	WAMANAGER_CICLO_DEPOSITO_FALDA_VUOTI_RUN:
		DirezioneXPositiva := TFDirezioneAssePositiva(Posizione_Attuale:=ModuleAX_X^.Ax^.Status.ActPosition,Posizione_Finale:=Mission^.XPlace);
		DirezioneXNegativa := NOT DirezioneXPositiva;
		(* Valuto se con l'asse X sono fuori dall'area delle colonne *)
		QuotaX_ConsensoRotazionePinza_Raggiunta := TFPinzaInFuoriIngombroColonne_DirezioneX(DirezioneXPositiva:=DirezioneXPositiva,
																							AsseInMoto:=ModuleAX_X^.Ax^.AxRef^.Status.Moving,
																							PosizioneAttuale:=ModuleAX_X^.Ax^.Status.ActPosition,
																							PosizioneColonna_X:=WorkFootprint^[5].X,  
																							IngombroColonna_X:=WorkFootprint^[5].XDim,
																							IngombroPinza_X:=IngombroX);
				IF CalcolaIngombro THEN
			CalcolaIngombro := FALSE;
			(* Definisco il tipo di area in cui si trova a lavorare il pallettizzatore *)
			AreaInLavoroPositiva := FALSE;
			AreaInLavoroNegativa := FALSE;
			AreaInLavoroPositivaNegativa := FALSE; 
			
			IF (WorkArea^[Mission^.PPlace].X >= (WorkFootprint^[5].X + WorkFootprint^[5].XDim)) AND 		//se la piazzola di prelievo è nella campata POSITIVA
				(ModuleAX_X^.Ax^.Status.ActPosition >= (WorkFootprint^[5].X + WorkFootprint^[5].XDim)) THEN // Se la posizione attuale è nella campata POSITIVA
					AreaInLavoroPositivaNegativa := FALSE; 
					AreaInLavoroPositiva := TRUE;
			ELSIF (WorkArea^[Mission^.PPlace].X <= WorkFootprint^[5].X) AND 			//se la piazzola di prelievo è nella campata NEGATIVA
				(ModuleAX_X^.Ax^.Status.ActPosition <= WorkFootprint^[5].X) THEN 		// Se la posizione attuale è nella campata NEGATIVA
					AreaInLavoroPositivaNegativa := FALSE; 
					AreaInLavoroNegativa := TRUE;
			ELSE
				AreaInLavoroPositivaNegativa := TRUE;
			END_IF
			
			(**************************************************************************************************************************************************)
			(* Ingombro ottimizzato della pinza sul punto di prelievo *)
			(**************************************************************************************************************************************************)
			IngombroOttimizzatoX_InPuntoDiPrelievo := ABS(IngombroSuperficialePinzaMAX * SIN(deg_to_rad((ATAN(Larghezza/Lunghezza)*1/0.017+ Mission^.JPick))));
			IngombroOttimizzatoY_InPuntoDiPrelievo := ABS(IngombroSuperficialePinzaMAX * COS(deg_to_rad((ATAN(Larghezza/Lunghezza)*1/0.017+ Mission^.JPick))));
			(**************************************************************************************************************************************************)
			(* Ingombro ottimizzato della pinza sul punto di deposito *)
			(**************************************************************************************************************************************************)
			IngombroOttimizzatoX_InPuntoDiDeposito := ABS(IngombroSuperficialePinzaMAX * SIN(deg_to_rad((ATAN(Larghezza/Lunghezza)*1/0.017+ Mission^.JPlace))));
			IngombroOttimizzatoY_InPuntoDiDeposito := ABS(IngombroSuperficialePinzaMAX * COS(deg_to_rad((ATAN(Larghezza/Lunghezza)*1/0.017+ Mission^.JPlace))));
						
			(**************************************************************************************************************************************************)
			(**************************************************************************************************************************************************)
			(* Valuto la direzione della X *)
			DirezioneXPositiva := TFDirezioneAssePositiva(Posizione_Attuale:=ModuleAX_X^.Ax^.Status.ActPosition,Posizione_Finale:=Mission^.XPlace);
			DirezioneXNegativa := NOT DirezioneXPositiva;
							
			(**************************************************************************************************************************************************)
			(* Ingombro MASSIMO della pinza durante il transito *)
			(**************************************************************************************************************************************************)
			//Calcolo ingombro attuale
			IF NOT TFAsseInFinestra(Posizione_Attuale:=ModuleAx_J^.Ax^.AxRef^.NcToPlc.ActPos,Posizione_Finale:=Mission^.JPlace,FinestraDiControllo:=5)  THEN //Se la pinza non è già nella finestra di destinazione 
				(* Calcolo l'ingombro massimo che assume durante il ciclo di lavoro nelle direzioni X e Y *)
				TFCalcoloIngombroOttimizzatoPinza(  Quota_RotazioneAttuale			:= ModuleAx_J^.Ax^.AxRef^.NcToPlc.ActPos,
													Quota_RotazioneDestinazione		:= Mission^.JPlace,
													IngombroSuperficialePinzaMAX	:= IngombroSuperficialePinzaMAX,
													Lunghezza						:= Larghezza,
													Larghezza						:= Lunghezza,
													IngombroOttimizzatoX_InTransito	=> IngombroOttimizzatoX_InTransito,
													IngombroOttimizzatoY_InTransito	=> IngombroOttimizzatoY_InTransito);
			ELSE
				IngombroOttimizzatoX_InTransito := ABS(IngombroSuperficialePinzaMAX * SIN(deg_to_rad((ATAN(Larghezza/Lunghezza)*1/0.017+ ModuleAx_J^.Ax^.AxRef^.NcToPlc.ActPos)))); //Ingombro Attuale direzione X
				IngombroOttimizzatoY_InTransito := ABS(IngombroSuperficialePinzaMAX * COS(deg_to_rad((ATAN(Larghezza/Lunghezza)*1/0.017+ ModuleAx_J^.Ax^.AxRef^.NcToPlc.ActPos)))); //Ingombro Attuale direzione Y		
			END_IF
			(* Valutazione colonne in base al verso del pallettizzatore: verso stabilito guardando il pallettizzatore con la linea alle spalle *)
			CASE VERSO_PALLETTIZZATORE OF
				PALLETTIZZATORE_DX :
									TFCalcolaQuotaIngombroColonne(	QuotaY_ColonnaDX						:= WorkFootprint^[6].Y, //DX
																	QuotaY_ColonnaSX						:= WorkFootprint^[5].Y, //SX
																	QuotaAttualeAsse						:= ModuleAX_Y^.Ax^.AxRef^.NcToPlc.ActPos,
																	IngombroOttimizzatoY_InTransito         := IngombroOttimizzatoY_InTransito,
																	OffsetSicurezza_Y						:= OffsetSicurezza_Y,
																	QuotaDestinazioneAsse					:= Mission^.YPlace,
																	Pinza_InIngombroColonne_Attuale 		=> Pinza_InIngombroColonne_Attuale,
																	Pinza_InIngombroColonne_Destinazione 	=> Pinza_InIngombroColonne_Destinazione,
																	QuotaFuoriIngombro_Attuale_Y 			=> QuotaFuoriIngombro_Attuale_Y,
																	QuotaFuoriIngombro_Destinazione_Y 		=> QuotaFuoriIngombro_Destinazione_Y);
																	
				PALLETTIZZATORE_SX :
									TFCalcolaQuotaIngombroColonne(	QuotaY_ColonnaDX						:= WorkFootprint^[6].Y, //DX
																	QuotaY_ColonnaSX						:= WorkFootprint^[5].Y, //SX
																	QuotaAttualeAsse						:= ModuleAX_Y^.Ax^.AxRef^.NcToPlc.ActPos,
																	OffsetSicurezza_Y						:= OffsetSicurezza_Y,
																	IngombroOttimizzatoY_InTransito         := IngombroOttimizzatoY_InTransito,
																	QuotaDestinazioneAsse					:= Mission^.YPlace,
																	Pinza_InIngombroColonne_Attuale 		=> Pinza_InIngombroColonne_Attuale,
																	Pinza_InIngombroColonne_Destinazione 	=> Pinza_InIngombroColonne_Destinazione,
																	QuotaFuoriIngombro_Attuale_Y 			=> QuotaFuoriIngombro_Attuale_Y,
																	QuotaFuoriIngombro_Destinazione_Y 		=> QuotaFuoriIngombro_Destinazione_Y);
			END_CASE
			
			(* Setto la quota di fuori ingombro che la pinza dovrà assumere durante la traslazione per evitare la collisione con le colonne *)	
			QuotaFuoriIngombroColonne_Y := MAX(QuotaFuoriIngombro_Attuale_Y,QuotaFuoriIngombro_Destinazione_Y);
					
			(* Se sono in ingombro nella posizione attuale o nella posizione di destinazione, devo andare fuori-ingombro con la Y *)
			IF (Pinza_InIngombroColonne_Attuale OR Pinza_InIngombroColonne_Destinazione) THEN 
				IF (AsseXInFinestraDiRiposo AND AsseYInFinestraDiRiposo AND AsseJInFinestraDiRiposo) THEN //Se sono in finestra di riposo con tutti gli assi non devo andare fuori-ingombro con la Y
					FuoriIngombroYNecessarioTMP := FALSE;
				ELSE
					FuoriIngombroYNecessarioTMP := TRUE;
				END_IF
			ELSE
				FuoriIngombroYNecessarioTMP := FALSE;
			END_IF
		END_IF
								
	//WAMANAGER_CICLO_DEPOSITO_FALDA_VUOTI_END:
	//	CalcolaIngombro := TRUE;	
	*)
	WAMANAGER_CICLO_FALDA_INIT:
		CalcolaIngombro := TRUE;	
	
	WAMANAGER_CICLO_PRELIEVO_FALDA_RUN:
		DirezioneXPositiva := TFDirezioneAssePositiva(Posizione_Attuale:=ModuleAX_X^.Ax^.Status.ActPosition,Posizione_Finale:=Mission^.XPick);
		DirezioneXNegativa := NOT DirezioneXPositiva;
		(* Valuto se con l'asse X sono fuori dall'area delle colonne *)
		(*QuotaX_ConsensoRotazionePinza_Raggiunta := TFPinzaInFuoriIngombroColonne_DirezioneX(DirezioneXPositiva:=DirezioneXPositiva,
																							AsseInMoto:=ModuleAX_X^.Ax^.AxRef^.Status.Moving,
																							PosizioneAttuale:=ModuleAX_X^.Ax^.Status.ActPosition,
																							PosizioneColonna_X:=WorkFootprint^[5].X,  
																							IngombroColonna_X:=WorkFootprint^[5].XDim,
																							IngombroPinza_X:=IngombroX);*)
																							
		IF CalcolaIngombro THEN
			CalcolaIngombro := FALSE;
			(* Definisco il tipo di area in cui si trova a lavorare il pallettizzatore *)
			AreaInLavoroPositiva := FALSE;
			AreaInLavoroNegativa := FALSE;
			AreaInLavoroPositivaNegativa := FALSE; 
			
			IF (WorkArea^[Mission^.PPick].X >= (WorkFootprint^[5].X + WorkFootprint^[5].XDim)) AND 				//se la piazzola di prelievo è nella campata POSITIVA
				(ModuleAX_X^.Ax^.Status.ActPosition >= (WorkFootprint^[5].X + WorkFootprint^[5].XDim)) THEN // Se la posizione attuale è nella campata POSITIVA
					AreaInLavoroPositiva := TRUE;
			ELSIF (WorkArea^[Mission^.PPick].X <= WorkFootprint^[5].X) AND 			//se la piazzola di prelievo è nella campata NEGATIVA
				(ModuleAX_X^.Ax^.Status.ActPosition <= WorkFootprint^[5].X) THEN 		// Se la posizione attuale è nella campata NEGATIVA
					AreaInLavoroNegativa := TRUE;
			ELSE
				AreaInLavoroPositivaNegativa := TRUE;
			END_IF
			(**************************************************************************************************************************************************)
			(* Ingombro ottimizzato della pinza sul punto di prelievo *)
			(**************************************************************************************************************************************************)
			(*IngombroOttimizzatoX_InPuntoDiPrelievo := ABS(IngombroSuperficialePinzaMAX * SIN(deg_to_rad((ATAN(Larghezza/Lunghezza)*1/0.017+ Mission^.JPick))));
			IngombroOttimizzatoY_InPuntoDiPrelievo := ABS(IngombroSuperficialePinzaMAX * COS(deg_to_rad((ATAN(Larghezza/Lunghezza)*1/0.017+ Mission^.JPick))));
			(**************************************************************************************************************************************************)
			(* Ingombro ottimizzato della pinza sul punto di deposito *)
			(**************************************************************************************************************************************************)
			IngombroOttimizzatoX_InPuntoDiDeposito := ABS(IngombroSuperficialePinzaMAX * SIN(deg_to_rad((ATAN(Larghezza/Lunghezza)*1/0.017+ Mission^.JPlace))));
			IngombroOttimizzatoY_InPuntoDiDeposito := ABS(IngombroSuperficialePinzaMAX * COS(deg_to_rad((ATAN(Larghezza/Lunghezza)*1/0.017+ Mission^.JPlace))));
			*)			
			(**************************************************************************************************************************************************)
			(**************************************************************************************************************************************************)
			(* Valuto la direzione della X *)
			DirezioneXPositiva := TFDirezioneAssePositiva(Posizione_Attuale:=ModuleAX_X^.Ax^.Status.ActPosition,Posizione_Finale:=Mission^.XPick);
			DirezioneXNegativa := NOT DirezioneXPositiva;
							
			(**************************************************************************************************************************************************)
			(* Ingombro MASSIMO della pinza durante il transito *)
			(**************************************************************************************************************************************************)
			//Calcolo ingombro attuale
			IF NOT TFAsseInFinestra(Posizione_Attuale:=ModuleAx_J^.Ax^.AxRef^.NcToPlc.ActPos,Posizione_Finale:=Mission^.JPick,FinestraDiControllo:=5)  THEN //Se la pinza non è già nella finestra di destinazione 
				(* Calcolo l'ingombro massimo che assume durante il ciclo di lavoro nelle direzioni X e Y *)
				(*TFCalcoloIngombroOttimizzatoPinza(  Quota_RotazioneAttuale			:= ModuleAx_J^.Ax^.AxRef^.NcToPlc.ActPos,
													Quota_RotazioneDestinazione		:= Mission^.JPick,
													IngombroSuperficialePinzaMAX	:= IngombroSuperficialePinzaMAX,
													Lunghezza						:= Larghezza,
													Larghezza						:= Lunghezza,
													IngombroOttimizzatoX_InTransito	=> IngombroOttimizzatoX_InTransito,
													IngombroOttimizzatoY_InTransito	=> IngombroOttimizzatoY_InTransito);*)
			ELSE;
				//IngombroOttimizzatoX_InTransito := ABS(IngombroSuperficialePinzaMAX * SIN(deg_to_rad((ATAN(Larghezza/Lunghezza)*1/0.017+ ModuleAx_J^.Ax^.AxRef^.NcToPlc.ActPos)))); //Ingombro Attuale direzione X
				//IngombroOttimizzatoY_InTransito := ABS(IngombroSuperficialePinzaMAX * COS(deg_to_rad((ATAN(Larghezza/Lunghezza)*1/0.017+ ModuleAx_J^.Ax^.AxRef^.NcToPlc.ActPos)))); //Ingombro Attuale direzione Y		
			END_IF
			(* Valutazione colonne in base al verso del pallettizzatore: verso stabilito guardando il pallettizzatore con la linea alle spalle *)
			CASE VERSO_PALLETTIZZATORE OF
				PALLETTIZZATORE_DX :
									TFCalcolaQuotaIngombroColonne(	QuotaY_ColonnaDX						:= WorkFootprint^[6].Y, //DX
																	QuotaY_ColonnaSX						:= WorkFootprint^[5].Y, //SX
																	QuotaAttualeAsse						:= ModuleAX_Y^.Ax^.AxRef^.NcToPlc.ActPos,
																	IngombroOttimizzatoY_InTransito         := IngombroOttimizzatoY_InTransito,
																	OffsetSicurezza_Y						:= OffsetSicurezza_Y,
																	QuotaDestinazioneAsse					:= Mission^.YPick,
																	Pinza_InIngombroColonne_Attuale 		=> Pinza_InIngombroColonne_Attuale,
																	Pinza_InIngombroColonne_Destinazione 	=> Pinza_InIngombroColonne_Destinazione,
																	QuotaFuoriIngombro_Attuale_Y 			=> QuotaFuoriIngombro_Attuale_Y,
																	QuotaFuoriIngombro_Destinazione_Y 		=> QuotaFuoriIngombro_Destinazione_Y);
																	
				PALLETTIZZATORE_SX :
									TFCalcolaQuotaIngombroColonne(	QuotaY_ColonnaDX						:= WorkFootprint^[6].Y, //DX
																	QuotaY_ColonnaSX						:= WorkFootprint^[5].Y, //SX
																	QuotaAttualeAsse						:= ModuleAX_Y^.Ax^.AxRef^.NcToPlc.ActPos,
																	OffsetSicurezza_Y						:= OffsetSicurezza_Y,
																	IngombroOttimizzatoY_InTransito         := IngombroOttimizzatoY_InTransito,
																	QuotaDestinazioneAsse					:= Mission^.YPick,
																	Pinza_InIngombroColonne_Attuale 		=> Pinza_InIngombroColonne_Attuale,
																	Pinza_InIngombroColonne_Destinazione 	=> Pinza_InIngombroColonne_Destinazione,
																	QuotaFuoriIngombro_Attuale_Y 			=> QuotaFuoriIngombro_Attuale_Y,
																	QuotaFuoriIngombro_Destinazione_Y 		=> QuotaFuoriIngombro_Destinazione_Y);
			END_CASE
			
			(* Setto la quota di fuori ingombro che la pinza dovrà assumere durante la traslazione per evitare la collisione con le colonne *)	
			QuotaFuoriIngombroColonne_Y := QuotaFuoriIngombro_Attuale_Y;
					
			(* Se sono in ingombro nella posizione attuale o nella posizione di destinazione, devo andare fuori-ingombro con la Y *)
			IF (Pinza_InIngombroColonne_Attuale OR Pinza_InIngombroColonne_Destinazione) THEN 
				IF (AsseXInFinestraDiRiposo AND AsseYInFinestraDiRiposo AND AsseJInFinestraDiRiposo) THEN //Se sono in finestra di riposo con tutti gli assi non devo andare fuori-ingombro con la Y
					FuoriIngombroYNecessarioTMP := FALSE;
				ELSE
					FuoriIngombroYNecessarioTMP := TRUE;
				END_IF
			ELSE
				FuoriIngombroYNecessarioTMP := FALSE;
			END_IF
		END_IF	
																
	WAMANAGER_CICLO_PRELIEVO_FALDA_END:
		CalcolaIngombro := TRUE;	
			
	WAMANAGER_CICLO_DEPOSITO_FALDA_RUN:
		DirezioneXPositiva := TFDirezioneAssePositiva(Posizione_Attuale:=ModuleAX_X^.Ax^.Status.ActPosition,Posizione_Finale:=Mission^.XPlace);
		DirezioneXNegativa := NOT DirezioneXPositiva;
		(* Valuto se con l'asse X sono fuori dall'area delle colonne *)
		(*QuotaX_ConsensoRotazionePinza_Raggiunta := TFPinzaInFuoriIngombroColonne_DirezioneX(DirezioneXPositiva:=DirezioneXPositiva,
																							AsseInMoto:=ModuleAX_X^.Ax^.AxRef^.Status.Moving,
																							PosizioneAttuale:=ModuleAX_X^.Ax^.Status.ActPosition,
																							PosizioneColonna_X:=WorkFootprint^[5].X,  
																							IngombroColonna_X:=WorkFootprint^[5].XDim,
																							IngombroPinza_X:=IngombroX);*)
																							
		IF (WorkArea^[Mission^.PPlace].X >= (WorkFootprint^[5].X + WorkFootprint^[5].XDim)) AND 				//se la piazzola di prelievo è nella campata POSITIVA
			(ModuleAX_X^.Ax^.Status.ActPosition >= (WorkFootprint^[5].X + WorkFootprint^[5].XDim)) THEN // Se la posizione attuale è nella campata POSITIVA
				AreaInLavoroPositiva := TRUE;
		ELSIF (WorkArea^[Mission^.PPlace].X <= WorkFootprint^[5].X) AND 			//se la piazzola di prelievo è nella campata NEGATIVA
			(ModuleAX_X^.Ax^.Status.ActPosition <= WorkFootprint^[5].X) THEN 		// Se la posizione attuale è nella campata NEGATIVA
				AreaInLavoroNegativa := TRUE;
		ELSE
			AreaInLavoroPositivaNegativa := TRUE;
		END_IF
		
		IF CalcolaIngombro THEN
			CalcolaIngombro := FALSE;
			(* Definisco il tipo di area in cui si trova a lavorare il pallettizzatore *)
			AreaInLavoroPositiva := FALSE;
			AreaInLavoroNegativa := FALSE;
			AreaInLavoroPositivaNegativa := TRUE; 
			
			(**************************************************************************************************************************************************)
			(* Ingombro ottimizzato della pinza sul punto di prelievo *)
			(**************************************************************************************************************************************************)
		(*	IngombroOttimizzatoX_InPuntoDiPrelievo := ABS(IngombroSuperficialePinzaMAX * SIN(deg_to_rad((ATAN(Larghezza/Lunghezza)*1/0.017+ Mission^.JPick))));
			IngombroOttimizzatoY_InPuntoDiPrelievo := ABS(IngombroSuperficialePinzaMAX * COS(deg_to_rad((ATAN(Larghezza/Lunghezza)*1/0.017+ Mission^.JPick))));
			(**************************************************************************************************************************************************)
			(* Ingombro ottimizzato della pinza sul punto di deposito *)
			(**************************************************************************************************************************************************)
			IngombroOttimizzatoX_InPuntoDiDeposito := ABS(IngombroSuperficialePinzaMAX * SIN(deg_to_rad((ATAN(Larghezza/Lunghezza)*1/0.017+ Mission^.JPlace))));
			IngombroOttimizzatoY_InPuntoDiDeposito := ABS(IngombroSuperficialePinzaMAX * COS(deg_to_rad((ATAN(Larghezza/Lunghezza)*1/0.017+ Mission^.JPlace))));
			*)			
			(**************************************************************************************************************************************************)
			(**************************************************************************************************************************************************)
			(* Valuto la direzione della X *)
			DirezioneXPositiva := TFDirezioneAssePositiva(Posizione_Attuale:=ModuleAX_X^.Ax^.Status.ActPosition,Posizione_Finale:=Mission^.XPlace);
			DirezioneXNegativa := NOT DirezioneXPositiva;
							
			(**************************************************************************************************************************************************)
			(* Ingombro MASSIMO della pinza durante il transito *)
			(**************************************************************************************************************************************************)
			//Calcolo ingombro attuale
			IF NOT TFAsseInFinestra(Posizione_Attuale:=ModuleAx_J^.Ax^.AxRef^.NcToPlc.ActPos,Posizione_Finale:=Mission^.JPlace,FinestraDiControllo:=5)  THEN //Se la pinza non è già nella finestra di destinazione 
				(* Calcolo l'ingombro massimo che assume durante il ciclo di lavoro nelle direzioni X e Y *)
				(*TFCalcoloIngombroOttimizzatoPinza(  Quota_RotazioneAttuale			:= ModuleAx_J^.Ax^.AxRef^.NcToPlc.ActPos,
													Quota_RotazioneDestinazione		:= Mission^.JPlace,
													IngombroSuperficialePinzaMAX	:= IngombroSuperficialePinzaMAX,
													Lunghezza						:= Larghezza,
													Larghezza						:= Lunghezza,
													IngombroOttimizzatoX_InTransito	=> IngombroOttimizzatoX_InTransito,
													IngombroOttimizzatoY_InTransito	=> IngombroOttimizzatoY_InTransito);*)
			ELSE;
				//IngombroOttimizzatoX_InTransito := ABS(IngombroSuperficialePinzaMAX * SIN(deg_to_rad((ATAN(Larghezza/Lunghezza)*1/0.017+ ModuleAx_J^.Ax^.AxRef^.NcToPlc.ActPos)))); //Ingombro Attuale direzione X
				//IngombroOttimizzatoY_InTransito := ABS(IngombroSuperficialePinzaMAX * COS(deg_to_rad((ATAN(Larghezza/Lunghezza)*1/0.017+ ModuleAx_J^.Ax^.AxRef^.NcToPlc.ActPos)))); //Ingombro Attuale direzione Y		
			END_IF
			(* Valutazione colonne in base al verso del pallettizzatore: verso stabilito guardando il pallettizzatore con la linea alle spalle *)
			CASE VERSO_PALLETTIZZATORE OF
				PALLETTIZZATORE_DX :
									TFCalcolaQuotaIngombroColonne(	QuotaY_ColonnaDX						:= WorkFootprint^[6].Y, //DX
																	QuotaY_ColonnaSX						:= WorkFootprint^[5].Y, //SX
																	QuotaAttualeAsse						:= ModuleAX_Y^.Ax^.AxRef^.NcToPlc.ActPos,
																	IngombroOttimizzatoY_InTransito         := IngombroOttimizzatoY_InTransito,
																	OffsetSicurezza_Y						:= OffsetSicurezza_Y,
																	QuotaDestinazioneAsse					:= Mission^.YPlace,
																	Pinza_InIngombroColonne_Attuale 		=> Pinza_InIngombroColonne_Attuale,
																	Pinza_InIngombroColonne_Destinazione 	=> Pinza_InIngombroColonne_Destinazione,
																	QuotaFuoriIngombro_Attuale_Y 			=> QuotaFuoriIngombro_Attuale_Y,
																	QuotaFuoriIngombro_Destinazione_Y 		=> QuotaFuoriIngombro_Destinazione_Y);
																	
				PALLETTIZZATORE_SX :
									TFCalcolaQuotaIngombroColonne(	QuotaY_ColonnaDX						:= WorkFootprint^[6].Y, //DX
																	QuotaY_ColonnaSX						:= WorkFootprint^[5].Y, //SX
																	QuotaAttualeAsse						:= ModuleAX_Y^.Ax^.AxRef^.NcToPlc.ActPos,
																	OffsetSicurezza_Y						:= OffsetSicurezza_Y,
																	IngombroOttimizzatoY_InTransito         := IngombroOttimizzatoY_InTransito,
																	QuotaDestinazioneAsse					:= Mission^.YPlace,
																	Pinza_InIngombroColonne_Attuale 		=> Pinza_InIngombroColonne_Attuale,
																	Pinza_InIngombroColonne_Destinazione 	=> Pinza_InIngombroColonne_Destinazione,
																	QuotaFuoriIngombro_Attuale_Y 			=> QuotaFuoriIngombro_Attuale_Y,
																	QuotaFuoriIngombro_Destinazione_Y 		=> QuotaFuoriIngombro_Destinazione_Y);
			END_CASE
			
			(* Setto la quota di fuori ingombro che la pinza dovrà assumere durante la traslazione per evitare la collisione con le colonne *)	
			QuotaFuoriIngombroColonne_Y := QuotaFuoriIngombro_Attuale_Y;
					
			(* Se sono in ingombro nella posizione attuale o nella posizione di destinazione, devo andare fuori-ingombro con la Y *)
			IF (Pinza_InIngombroColonne_Attuale OR Pinza_InIngombroColonne_Destinazione) THEN 
				IF (AsseXInFinestraDiRiposo AND AsseYInFinestraDiRiposo AND AsseJInFinestraDiRiposo) THEN //Se sono in finestra di riposo con tutti gli assi non devo andare fuori-ingombro con la Y
					FuoriIngombroYNecessarioTMP := FALSE;
				ELSE
					FuoriIngombroYNecessarioTMP := TRUE;
				END_IF
			ELSE
				FuoriIngombroYNecessarioTMP := FALSE;
			END_IF
		END_IF
			
	WAMANAGER_CICLO_DEPOSITO_FALDA_END:
		CalcolaIngombro := TRUE;	
(*
	WAMANAGER_CICLO_PACCO_INIT:
		CalcolaIngombro := TRUE;	
	
	WAMANAGER_CICLO_PRELIEVO_PACCO_RUN:
		DirezioneXPositiva := TFDirezioneAssePositiva(Posizione_Attuale:=ModuleAX_X^.Ax^.Status.ActPosition,Posizione_Finale:=Mission^.XPick);
		DirezioneXNegativa := NOT DirezioneXPositiva;
		(* Valuto se con l'asse X sono fuori dall'area delle colonne *)
		QuotaX_ConsensoRotazionePinza_Raggiunta := TFPinzaInFuoriIngombroColonne_DirezioneX(DirezioneXPositiva:=DirezioneXPositiva,
																							AsseInMoto:=ModuleAX_X^.Ax^.AxRef^.Status.Moving,
																							PosizioneAttuale:=ModuleAX_X^.Ax^.Status.ActPosition,
																							PosizioneColonna_X:=WorkFootprint^[5].X,  
																							IngombroColonna_X:=WorkFootprint^[5].XDim,
																							IngombroPinza_X:=IngombroX);																				
		
		IF CalcolaIngombro THEN
			CalcolaIngombro := FALSE;
			(* Definisco il tipo di area in cui si trova a lavorare il pallettizzatore *)
			AreaInLavoroPositiva := FALSE;
			AreaInLavoroNegativa := FALSE;
			AreaInLavoroPositivaNegativa := TRUE; 
			
			(**************************************************************************************************************************************************)
			(* Ingombro ottimizzato della pinza sul punto di prelievo *)
			(**************************************************************************************************************************************************)
			IngombroOttimizzatoX_InPuntoDiPrelievo := ABS(IngombroSuperficialePinzaMAX * SIN(deg_to_rad((ATAN(Larghezza/Lunghezza)*1/0.017+ Mission^.JPick))));
			IngombroOttimizzatoY_InPuntoDiPrelievo := ABS(IngombroSuperficialePinzaMAX * COS(deg_to_rad((ATAN(Larghezza/Lunghezza)*1/0.017+ Mission^.JPick))));
			(**************************************************************************************************************************************************)
			(* Ingombro ottimizzato della pinza sul punto di deposito *)
			(**************************************************************************************************************************************************)
			IngombroOttimizzatoX_InPuntoDiDeposito := ABS(IngombroSuperficialePinzaMAX * SIN(deg_to_rad((ATAN(Larghezza/Lunghezza)*1/0.017+ Mission^.JPlace))));
			IngombroOttimizzatoY_InPuntoDiDeposito := ABS(IngombroSuperficialePinzaMAX * COS(deg_to_rad((ATAN(Larghezza/Lunghezza)*1/0.017+ Mission^.JPlace))));
						
			(**************************************************************************************************************************************************)
			(**************************************************************************************************************************************************)
			(* Valuto la direzione della X *)
			DirezioneXPositiva := TFDirezioneAssePositiva(Posizione_Attuale:=ModuleAX_X^.Ax^.Status.ActPosition,Posizione_Finale:=Mission^.XPick);
			DirezioneXNegativa := NOT DirezioneXPositiva;
							
			(**************************************************************************************************************************************************)
			(* Ingombro MASSIMO della pinza durante il transito *)
			(**************************************************************************************************************************************************)
			//Calcolo ingombro attuale
			IF NOT TFAsseInFinestra(Posizione_Attuale:=ModuleAx_J^.Ax^.AxRef^.NcToPlc.ActPos,Posizione_Finale:=Mission^.JPick,FinestraDiControllo:=5)  THEN //Se la pinza non è già nella finestra di destinazione 
				(* Calcolo l'ingombro massimo che assume durante il ciclo di lavoro nelle direzioni X e Y *)
				TFCalcoloIngombroOttimizzatoPinza(  Quota_RotazioneAttuale			:= ModuleAx_J^.Ax^.AxRef^.NcToPlc.ActPos,
													Quota_RotazioneDestinazione		:= Mission^.JPick,
													IngombroSuperficialePinzaMAX	:= IngombroSuperficialePinzaMAX,
													Lunghezza						:= Larghezza,
													Larghezza						:= Lunghezza,
													IngombroOttimizzatoX_InTransito	=> IngombroOttimizzatoX_InTransito,
													IngombroOttimizzatoY_InTransito	=> IngombroOttimizzatoY_InTransito);
			ELSE
				IngombroOttimizzatoX_InTransito := ABS(IngombroSuperficialePinzaMAX * SIN(deg_to_rad((ATAN(Larghezza/Lunghezza)*1/0.017+ ModuleAx_J^.Ax^.AxRef^.NcToPlc.ActPos)))); //Ingombro Attuale direzione X
				IngombroOttimizzatoY_InTransito := ABS(IngombroSuperficialePinzaMAX * COS(deg_to_rad((ATAN(Larghezza/Lunghezza)*1/0.017+ ModuleAx_J^.Ax^.AxRef^.NcToPlc.ActPos)))); //Ingombro Attuale direzione Y		
			END_IF
			(* Valutazione colonne in base al verso del pallettizzatore: verso stabilito guardando il pallettizzatore con la linea alle spalle *)
			CASE VERSO_PALLETTIZZATORE OF
				PALLETTIZZATORE_DX :
									TFCalcolaQuotaIngombroColonne(	QuotaY_ColonnaDX						:= WorkFootprint^[6].Y, //DX
																	QuotaY_ColonnaSX						:= WorkFootprint^[5].Y, //SX
																	QuotaAttualeAsse						:= ModuleAX_Y^.Ax^.AxRef^.NcToPlc.ActPos,
																	IngombroOttimizzatoY_InTransito         := IngombroOttimizzatoY_InTransito,
																	OffsetSicurezza_Y						:= OffsetSicurezza_Y,
																	QuotaDestinazioneAsse					:= Mission^.YPick,
																	Pinza_InIngombroColonne_Attuale 		=> Pinza_InIngombroColonne_Attuale,
																	Pinza_InIngombroColonne_Destinazione 	=> Pinza_InIngombroColonne_Destinazione,
																	QuotaFuoriIngombro_Attuale_Y 			=> QuotaFuoriIngombro_Attuale_Y,
																	QuotaFuoriIngombro_Destinazione_Y 		=> QuotaFuoriIngombro_Destinazione_Y);
																	
				PALLETTIZZATORE_SX :
									TFCalcolaQuotaIngombroColonne(	QuotaY_ColonnaDX						:= WorkFootprint^[6].Y, //DX
																	QuotaY_ColonnaSX						:= WorkFootprint^[5].Y, //SX
																	QuotaAttualeAsse						:= ModuleAX_Y^.Ax^.AxRef^.NcToPlc.ActPos,
																	OffsetSicurezza_Y						:= OffsetSicurezza_Y,
																	IngombroOttimizzatoY_InTransito         := IngombroOttimizzatoY_InTransito,
																	QuotaDestinazioneAsse					:= Mission^.YPick,
																	Pinza_InIngombroColonne_Attuale 		=> Pinza_InIngombroColonne_Attuale,
																	Pinza_InIngombroColonne_Destinazione 	=> Pinza_InIngombroColonne_Destinazione,
																	QuotaFuoriIngombro_Attuale_Y 			=> QuotaFuoriIngombro_Attuale_Y,
																	QuotaFuoriIngombro_Destinazione_Y 		=> QuotaFuoriIngombro_Destinazione_Y);
			END_CASE
			
			(* Setto la quota di fuori ingombro che la pinza dovrà assumere durante la traslazione per evitare la collisione con le colonne *)	
			QuotaFuoriIngombroColonne_Y := QuotaFuoriIngombro_Attuale_Y;
					
			(* Se sono in ingombro nella posizione attuale o nella posizione di destinazione, devo andare fuori-ingombro con la Y *)
			IF (Pinza_InIngombroColonne_Attuale OR Pinza_InIngombroColonne_Destinazione) THEN 
				IF (AsseXInFinestraDiRiposo AND AsseYInFinestraDiRiposo AND AsseJInFinestraDiRiposo) THEN //Se sono in finestra di riposo con tutti gli assi non devo andare fuori-ingombro con la Y
					FuoriIngombroYNecessarioTMP := FALSE;
				ELSE
					FuoriIngombroYNecessarioTMP := TRUE;
				END_IF
			ELSE
				FuoriIngombroYNecessarioTMP := FALSE;
			END_IF
		END_IF
		
	WAMANAGER_CICLO_PRELIEVO_PACCO_END:
		CalcolaIngombro := TRUE;	
		
	WAMANAGER_CICLO_DEPOSITO_PACCO_RUN:
		DirezioneXPositiva := TFDirezioneAssePositiva(Posizione_Attuale:=ModuleAX_X^.Ax^.Status.ActPosition,Posizione_Finale:=Mission^.XPlace);
		DirezioneXNegativa := NOT DirezioneXPositiva;
		
		
		(* Larhezza Pick Point + Pacco *)
		(*IF WorkPickPointState^[1].XDim >= WorkPickPointDimension[1].XDim THEN
			LarghezzaPickPoint := WorkPickPointState^[1].XDim;
		else
			LarghezzaPickPoint := WorkPickPointDimension[1].Xdim;
		END_IF*)
				
		(* Valuto se con l'asse X sono fuori dall'area delle colonne *)
		QuotaX_ConsensoRotazionePinza_Raggiunta := TFPinzaInFuoriIngombroColonne_DirezioneX(DirezioneXPositiva:=DirezioneXPositiva,
																							AsseInMoto:=ModuleAX_X^.Ax^.AxRef^.Status.Moving,
																							PosizioneAttuale:=ModuleAX_X^.Ax^.Status.ActPosition,
																							PosizioneColonna_X:=WorkFootprint^[5].X,  
																							IngombroColonna_X:=WorkFootprint^[5].XDim,
																							IngombroPinza_X:=IngombroX);
		
		(*IF (WorkPickPoint^[Mission^.PPick].Xh >= WorkArea^[Mission^.PPlace].X AND Mission^.JPickVO = 1) OR 	//se il punto di prelievo IN ORRIZZONTALE ha quota maggiore della piazzola di deposito e
			(WorkPickPoint^[Mission^.PPick].Xv >= WorkArea^[Mission^.PPlace].X AND Mission^.JPickVO = 0) THEN
			 AreaInLavoroNegativa := TRUE;
		ELSIF (WorkPickPoint^[Mission^.PPick].Xh <= WorkArea^[Mission^.PPlace].X AND Mission^.JPickVO = 1) OR 	//se il punto di prelievo IN ORRIZZONTALE ha quota maggiore della piazzola di deposito e
			(WorkPickPoint^[Mission^.PPick].Xv <= WorkArea^[Mission^.PPlace].X AND Mission^.JPickVO = 0) THEN
			 AreaInLavoroPositiva := TRUE;
		END_IF*)																					
		CASE TIPO_RIBALTINO OF

			RIBALTINO_DOPO_SQUADRO:
									(* Valutazione Fuoringombro lungo X della pinza rispetto al ribaltino + Pacco*)
									IF (ModuleAX_X^.Ax^.Status.ActPosition + IngombroX/ 2 <= WorkPickPoint^[Mission^.PPick].Xv - LarghezzaPickPoint/2 + 30) OR 
										(ModuleAX_X^.Ax^.Status.ActPosition - IngombroX/ 2 >= WorkPickPoint^[Mission^.PPick].Xv + LarghezzaPickPoint/2 - 30) THEN
											QuotaFUPRINGOMBROdaRIBALTINO_X_RAGGIUNTA := TRUE;
									ELSE
										QuotaFUPRINGOMBROdaRIBALTINO_X_RAGGIUNTA := FALSE;
									END_IF
									
			RIBALTINO_DIRETTO:
							   (* Valutazione Fuoringombro lungo X della pinza rispetto al ribaltino + Pacco*)
								IF (ModuleAX_X^.Ax^.Status.ActPosition + IngombroX/ 2 <= WorkPickPoint^[Mission^.PPick].Xv + 30) OR 
									(ModuleAX_X^.Ax^.Status.ActPosition - IngombroX/ 2 >= WorkPickPoint^[Mission^.PPick].Xv - 30) THEN
										QuotaFUPRINGOMBROdaRIBALTINO_X_RAGGIUNTA := TRUE;
								ELSE
									QuotaFUPRINGOMBROdaRIBALTINO_X_RAGGIUNTA := FALSE;
								END_IF
								
								(* Valutazione Fuoringombro lungo Y della pinza rispetto al ribaltino + Pacco*)
								IF (ModuleAX_Y^.Ax^.Status.ActPosition + IngombroY/ 2 <= WorkPickPoint^[Mission^.PPick].Yv - LarghezzaPickPoint/2 + 30) OR 
									(ModuleAX_Y^.Ax^.Status.ActPosition - IngombroY/ 2 >= WorkPickPoint^[Mission^.PPick].Yv + LarghezzaPickPoint/2 - 30) OR
									(ModuleAX_Y^.Ax^.Status.ActPosition + IngombroY/ 2 <= WorkPickPoint^[Mission^.PPick].Yh - LarghezzaPickPoint/2 + 30) OR 
									(ModuleAX_Y^.Ax^.Status.ActPosition - IngombroY/ 2 >= WorkPickPoint^[Mission^.PPick].Yh + LarghezzaPickPoint/2 - 30) THEN
										QuotaFUPRINGOMBROdaRIBALTINO_Y_RAGGIUNTA := TRUE;
								ELSE
									QuotaFUPRINGOMBROdaRIBALTINO_Y_RAGGIUNTA := FALSE;
								END_IF
		END_CASE																	
																							
		IF CalcolaIngombro THEN
			CalcolaIngombro := FALSE;
			(* Definisco il tipo di area in cui si trova a lavorare il pallettizzatore *)
			AreaInLavoroPositiva := FALSE;
			AreaInLavoroNegativa := FALSE;
			AreaInLavoroPositivaNegativa := TRUE; 
			
			(**************************************************************************************************************************************************)
			(* Ingombro ottimizzato della pinza sul punto di prelievo *)
			(**************************************************************************************************************************************************)
			IngombroOttimizzatoX_InPuntoDiPrelievo := ABS(IngombroSuperficialePinzaMAX * SIN(deg_to_rad((ATAN(Larghezza/Lunghezza)*1/0.017+ Mission^.JPick))));
			IngombroOttimizzatoY_InPuntoDiPrelievo := ABS(IngombroSuperficialePinzaMAX * COS(deg_to_rad((ATAN(Larghezza/Lunghezza)*1/0.017+ Mission^.JPick))));
			(**************************************************************************************************************************************************)
			(* Ingombro ottimizzato della pinza sul punto di deposito *)
			(**************************************************************************************************************************************************)
			IngombroOttimizzatoX_InPuntoDiDeposito := ABS(IngombroSuperficialePinzaMAX * SIN(deg_to_rad((ATAN(Larghezza/Lunghezza)*1/0.017+ Mission^.JPlace))));
			IngombroOttimizzatoY_InPuntoDiDeposito := ABS(IngombroSuperficialePinzaMAX * COS(deg_to_rad((ATAN(Larghezza/Lunghezza)*1/0.017+ Mission^.JPlace))));
						
			(**************************************************************************************************************************************************)
			(**************************************************************************************************************************************************)
			(* Valuto la direzione della X *)
			DirezioneXPositiva := TFDirezioneAssePositiva(Posizione_Attuale:=ModuleAX_X^.Ax^.Status.ActPosition,Posizione_Finale:=Mission^.XPlace);
			DirezioneXNegativa := NOT DirezioneXPositiva;
							
			(**************************************************************************************************************************************************)
			(* Ingombro MASSIMO della pinza durante il transito *)
			(**************************************************************************************************************************************************)
			//Calcolo ingombro attuale
			IF NOT TFAsseInFinestra(Posizione_Attuale:=ModuleAx_J^.Ax^.AxRef^.NcToPlc.ActPos,Posizione_Finale:=Mission^.JPlace,FinestraDiControllo:=5)  THEN //Se la pinza non è già nella finestra di destinazione 
				(* Calcolo l'ingombro massimo che assume durante il ciclo di lavoro nelle direzioni X e Y *)
				TFCalcoloIngombroOttimizzatoPinza(  Quota_RotazioneAttuale			:= ModuleAx_J^.Ax^.AxRef^.NcToPlc.ActPos,
													Quota_RotazioneDestinazione		:= Mission^.JPlace,
													IngombroSuperficialePinzaMAX	:= IngombroSuperficialePinzaMAX,
													Lunghezza						:= Larghezza,
													Larghezza						:= Lunghezza,
													IngombroOttimizzatoX_InTransito	=> IngombroOttimizzatoX_InTransito,
													IngombroOttimizzatoY_InTransito	=> IngombroOttimizzatoY_InTransito);
			ELSE
				IngombroOttimizzatoX_InTransito := ABS(IngombroSuperficialePinzaMAX * SIN(deg_to_rad((ATAN(Larghezza/Lunghezza)*1/0.017+ ModuleAx_J^.Ax^.AxRef^.NcToPlc.ActPos)))); //Ingombro Attuale direzione X
				IngombroOttimizzatoY_InTransito := ABS(IngombroSuperficialePinzaMAX * COS(deg_to_rad((ATAN(Larghezza/Lunghezza)*1/0.017+ ModuleAx_J^.Ax^.AxRef^.NcToPlc.ActPos)))); //Ingombro Attuale direzione Y		
			END_IF
			(* Valutazione colonne in base al verso del pallettizzatore: verso stabilito guardando il pallettizzatore con la linea alle spalle *)
			CASE VERSO_PALLETTIZZATORE OF
				PALLETTIZZATORE_DX :
									TFCalcolaQuotaIngombroColonne(	QuotaY_ColonnaDX						:= WorkFootprint^[6].Y, //DX
																	QuotaY_ColonnaSX						:= WorkFootprint^[5].Y, //SX
																	QuotaAttualeAsse						:= ModuleAX_Y^.Ax^.AxRef^.NcToPlc.ActPos,
																	IngombroOttimizzatoY_InTransito         := IngombroOttimizzatoY_InTransito,
																	OffsetSicurezza_Y						:= OffsetSicurezza_Y,
																	QuotaDestinazioneAsse					:= Mission^.YPlace,
																	Pinza_InIngombroColonne_Attuale 		=> Pinza_InIngombroColonne_Attuale,
																	Pinza_InIngombroColonne_Destinazione 	=> Pinza_InIngombroColonne_Destinazione,
																	QuotaFuoriIngombro_Attuale_Y 			=> QuotaFuoriIngombro_Attuale_Y,
																	QuotaFuoriIngombro_Destinazione_Y 		=> QuotaFuoriIngombro_Destinazione_Y);
																	
				PALLETTIZZATORE_SX :
									TFCalcolaQuotaIngombroColonne(	QuotaY_ColonnaDX						:= WorkFootprint^[6].Y, //DX
																	QuotaY_ColonnaSX						:= WorkFootprint^[5].Y, //SX
																	QuotaAttualeAsse						:= ModuleAX_Y^.Ax^.AxRef^.NcToPlc.ActPos,
																	OffsetSicurezza_Y						:= OffsetSicurezza_Y,
																	IngombroOttimizzatoY_InTransito         := IngombroOttimizzatoY_InTransito,
																	QuotaDestinazioneAsse					:= Mission^.YPlace,
																	Pinza_InIngombroColonne_Attuale 		=> Pinza_InIngombroColonne_Attuale,
																	Pinza_InIngombroColonne_Destinazione 	=> Pinza_InIngombroColonne_Destinazione,
																	QuotaFuoriIngombro_Attuale_Y 			=> QuotaFuoriIngombro_Attuale_Y,
																	QuotaFuoriIngombro_Destinazione_Y 		=> QuotaFuoriIngombro_Destinazione_Y);
			END_CASE
			
			(* Setto la quota di fuori ingombro che la pinza dovrà assumere durante la traslazione per evitare la collisione con le colonne *)	
			QuotaFuoriIngombroColonne_Y := QuotaFuoriIngombro_Attuale_Y;
					
			(* Se sono in ingombro nella posizione attuale o nella posizione di destinazione, devo andare fuori-ingombro con la Y *)
			IF (Pinza_InIngombroColonne_Attuale OR Pinza_InIngombroColonne_Destinazione) THEN 
				IF (AsseXInFinestraDiRiposo AND AsseYInFinestraDiRiposo AND AsseJInFinestraDiRiposo) THEN //Se sono in finestra di riposo con tutti gli assi non devo andare fuori-ingombro con la Y
					FuoriIngombroYNecessarioTMP := FALSE;
				ELSE
					FuoriIngombroYNecessarioTMP := TRUE;
				END_IF
			ELSE
				FuoriIngombroYNecessarioTMP := FALSE;
			END_IF
		END_IF
		
	WAMANAGER_CICLO_DEPOSITO_PACCO_END:
		CalcolaIngombro := TRUE;	*)
	
END_CASE

END_FUNCTION_BLOCK

// ---- POUs/TFPalletizerDataTF/NON_USATE/TFCalcoliFuoriIngombriColonne_old.TcPOU
FUNCTION TFCalcoliFuoriIngombriColonne_old : BOOL
VAR_INPUT
	Traiettoria : POINTER TO TFTraiettoria;
	WorkSpace : POINTER TO TFMachinePalletizer_WorkSpace;
	WorkFootprint : POINTER TO ARRAY [1..MAXFOOTPRINT] OF TFMachinePalletizer_WorkFootprint; //Ingombri
	WorkPickPoint : POINTER TO ARRAY [1..MAXPICKPOINT] OF TFMachinePalletizer_WorkPickPoint;
	WorkPickPointState : POINTER TO ARRAY [1..MAXPICKPOINT] OF TFMachinePalletizer_WorkPickPointState;
	WorkArea : POINTER TO ARRAY [1..MAXAREA] OF TFMachinePalletizer_WorkArea;
	WorkAreaState : POINTER TO ARRAY [1..MAXAREA] OF TFMachinePalletizer_WorkAreaState;
	Pallet : POINTER TO ARRAY [1..MAXPALLET] OF TFMachinePalletizer_Pallet;
	Layer : POINTER TO ARRAY [1..MAXLAYER] OF TFMachinePalletizer_Layer;
	Forming : POINTER TO ARRAY [1..MAXFORMING] OF TFMachinePalletizer_Forming;
	PickPlaceParameters	: POINTER TO TFMachinePalletizer_ParametersFromHMI;
	Mission : POINTER TO TFMachinePalletizer_Mission;
	
	WorkAreaManager : POINTER TO TFWorkAreaManager;
	ModuleAX_X : POINTER TO TFModulePalletizer_Ax;
	ModuleAX_Y : POINTER TO TFModulePalletizer_Ax;
	ModuleAX_Z : POINTER TO TFModulePalletizer_Ax;
	ModuleAX_J : POINTER TO TFModulePalletizer_Ax;
	ModuleAX_K : POINTER TO TFModulePalletizer_Ax;
	AbilitaAnticipoDinamico : BOOL;
	AbilitaCalcoloIngombroOttimizzato : BOOL := TRUE; //Abilitazione dell'utilizzo degli ingombri ottimizzati... calcoli in base all'angolo di rotazione della pinza
END_VAR
VAR
	f : INT;
	a : INT;
	P : INT;
	wa : int;
	waDXSX : INT;
	AltezzaDiIngombroArea : REAL;
	AltezzaDiIngombroOstacoli : REAL;
	AltezzaDiIngombroPuntiPrelievo : REAL;
	AssegnaQuote : BOOL;
	
	Lunghezza : REAL;
	Larghezza : REAL;
	IngombroSuperficialePinzaMAX : REAL;
	IngombroX : REAL;
	IngombroY : REAL;
	IngombroZ : REAL;
	IngombroOttimizzatoX : REAL;
	IngombroOttimizzatoY : REAL;
	
	IngombroVerticalePinzaMAX : REAL;
	IngombroVerticaleMaxElementi : REAL;
	//DirezioneXPositiva_Dep : BOOL;
	//DirezioneXNegativa_Dep : BOOL;
	//DirezioneXPositiva_Prel : BOOL;
	//DirezioneXNegativa_Prel : BOOL;
	DirezioneZPositiva : BOOL;
	DirezioneZNegativa : BOOL;
	DirezioneXNegativa : BOOL;
	DirezioneXPositiva : BOOL;
	
	
	WASX : UINT;
	WADX : UINT;
	WAPARTENZA : UINT;
	WADESTINAZIONE : UINT;
	LarghezzaPickPoint : REAL;
	
	
	FuoriIngombroYNecessarioTMP : BOOL;
	QuotaX_ConsensoRotazionePinza_RaggiuntaTMP : BOOL;
	ConsensoTraslazioneY_TraColonneTMP : BOOL;
	AsseXInFinestraDiPrelievoPaccoTMP : BOOL;
	AsseJInFinestraDiPrelievoPaccoTMP : BOOL;
	
	OffsetSicurezza_Y : real := 50;
	
	
	Pinza_InIngombroColonne_Partenza: BOOL; //Indica che la posizione della pinza è in ingombro colonne alla partenza del ciclo/ REAL TIME
	IngombroOttimizzatoY_Destinazione: LREAL;
	IngombroOttimizzatoX_Destinazione: LREAL;
	IngombroOttimizzatoX_InPuntoDiPrelievo: LREAL;
	IngombroOttimizzatoY_InPuntoDiPrelievo: LREAL;
	IngombroOttimizzatoY_InPuntoDiDeposito: LREAL;
	IngombroOttimizzatoX_InPuntoDiDeposito: LREAL;
	Pinza_InIngombroColonne_Attuale: BOOL;
	Pinza_InIngombroColonne_Destinazione: BOOL;
	AsseJInFinestraDiPrelievoPallet: BOOL;
	AsseXInFinestraDiPrelievoPallet: BOOL;
	AsseYInFinestraDiPrelievoPallet: BOOL;
	AsseXInFinestraDiRiposo: BOOL;
	AsseYInFinestraDiRiposo: BOOL;
	AsseJInFinestraDiRiposo: BOOL;
	AsseXInFinestraDiDestinazione: BOOL;
	AsseJInFinestraDiDestinazione: BOOL;
	AsseYInFinestraDiDestinazione: BOOL;
	IngombroOttimizzatoX_InTransito: LREAL;
	IngombroOttimizzatoY_InTransito: LREAL;
	Pinza_InIngombroColonne_Transito: BOOL;
	Angolo: INT;
	CalcolaIngombro: BOOL;
	AsseXInFinestraDiPrelievo: BOOL;
	AsseYInFinestraDiPrelievo: BOOL;
	AsseJInFinestraDiPrelievo: BOOL;
	
	QuotaFuoriIngombro_Attuale_Y 		: LREAL;
	QuotaFuoriIngombro_Prelievo_Y 		: LREAL;
	QuotaFuoriIngombro_Deposito_Y		: LREAL;
END_VAR

TFCalcoliFuoriIngombriColonne := FALSE;

FuoriIngombroYNecessarioTMP := TRUE;
////////////////////////////////////////////////////////////////////////////////////////////////////////////////////////////////////////////////////////////
///////////////////////////////////////////////////////////////////////////////////////////////////////////////////////////////////////////////////////////
(**************************************************************************************************************************************************)
(**************************************************************************************************************************************************)
(**************************************************************************************************************************************************)
(**************************************************************************************************************************************************)
(* Calcolo Dimensioni pinza *)
(**************************************************************************************************************************************************)
Larghezza :=  Dimensioni_Pinza.Larghezza;
Lunghezza :=  Dimensioni_Pinza.Lunghezza; //Fisso la lunghezza

(* Calcolo delle dimensioni della pinza in base al tipo di ciclo in corso *)
CASE WorkAreaManager^.State OF
	WAMANAGER_NOP,
	
	WAMANAGER_CICLO_RIPOSO_INIT,
		
	WAMANAGER_CICLO_RIPOSO_RUN:
		
		IF (Mission^.KPick > Lunghezza) THEN // Se l'apertura in prelievo è maggiore della lunghezza della pinza
			Lunghezza := Mission^.KPick;
		END_IF
		IF (Mission^.KPlace > Lunghezza) THEN // // Se l'apertura in deposito è maggiore della lunghezza della pinza 
			Lunghezza := Mission^.KPlace;
		END_IF
		
	WAMANAGER_CICLO_PRELIEVO_PALL_RUN:
		IF ModuleAX_K^.Ax^.Status.ActPosition >= Dimensioni_Pinza.Lunghezza THEN
			Lunghezza := ModuleAX_K^.Ax^.Status.ActPosition;
		ELSE
			Lunghezza := Dimensioni_Pinza.Lunghezza;
		END_IF
				
	WAMANAGER_CICLO_DEPOSITO_PALL_RUN:
		IF ModuleAX_K^.Ax^.Status.ActPosition >= Dimensioni_Pinza.Lunghezza THEN
			Lunghezza := ModuleAX_K^.Ax^.Status.ActPosition;
		ELSE
			Lunghezza := Dimensioni_Pinza.Lunghezza;
		END_IF
		Larghezza :=  Mission^.YDim;
	
	WAMANAGER_CICLO_PRELIEVO_FALDA_VUOTI_RUN:
		IF ModuleAX_K^.Ax^.Status.ActPosition >= Dimensioni_Pinza.Lunghezza THEN
			Lunghezza := ModuleAX_K^.Ax^.Status.ActPosition;
		ELSE
			Lunghezza := Dimensioni_Pinza.Lunghezza;
		END_IF
		Larghezza :=  Mission^.YDim;
						
	WAMANAGER_CICLO_DEPOSITO_FALDA_VUOTI_RUN:
		IF ModuleAX_K^.Ax^.Status.ActPosition >= Dimensioni_Pinza.Lunghezza THEN
			Lunghezza := ModuleAX_K^.Ax^.Status.ActPosition;
		ELSE
			Lunghezza := Dimensioni_Pinza.Lunghezza;
		END_IF
		Larghezza :=  Mission^.YDim;
									
	WAMANAGER_CICLO_PRELIEVO_FALDA_RUN:
		IF ModuleAX_K^.Ax^.Status.ActPosition >= Dimensioni_Pinza.Lunghezza THEN
			Lunghezza := ModuleAX_K^.Ax^.Status.ActPosition;
		ELSE
			Lunghezza := Dimensioni_Pinza.Lunghezza;
		END_IF
		Larghezza :=  Mission^.YDim;
					
	WAMANAGER_CICLO_DEPOSITO_FALDA_RUN:
		IF ModuleAX_K^.Ax^.Status.ActPosition >= Dimensioni_Pinza.Lunghezza THEN
			Lunghezza := ModuleAX_K^.Ax^.Status.ActPosition;
		ELSE
			Lunghezza := Dimensioni_Pinza.Lunghezza;
		END_IF
		Larghezza :=  Mission^.YDim;
				
	WAMANAGER_CICLO_PRELIEVO_PACCO_RUN:
		IF Mission^.JPickLT = 0 AND Mission^.JPickVO = 0 THEN // se longitudinale ( PARALLELO A X) e in verticale
			Larghezza :=  Mission^.ZDim;
			IF Mission^.XDim + PickPlaceParameters^.OffsetKPickPack >= Dimensioni_Pinza.Lunghezza THEN
				Lunghezza := Mission^.XDim + PickPlaceParameters^.OffsetKPickPack;
			ELSE
				Lunghezza := Dimensioni_Pinza.Lunghezza;
			END_IF
		ELSIF  Mission^.JPickLT = 0 AND  Mission^.JPickVO = 1 THEN	// se longitudinale ( PARALLELO A X) e in orrizzontale
			Larghezza :=  Mission^.YDim;
			IF Mission^.XDim + PickPlaceParameters^.OffsetKPickPack >= Dimensioni_Pinza.Lunghezza THEN
				Lunghezza := Mission^.XDim + PickPlaceParameters^.OffsetKPickPack;
			ELSE
				Lunghezza := Dimensioni_Pinza.Lunghezza;
			END_IF
		ELSIF  Mission^.JPickLT = 1 AND  Mission^.JPickVO = 0 THEN	// se trasversale ( PARALLELO A Y) e in verticale
			Larghezza :=  Mission^.XDim;
			IF Mission^.ZDim + PickPlaceParameters^.OffsetKPickPack >= Dimensioni_Pinza.Lunghezza THEN
				Lunghezza := Mission^.ZDim + PickPlaceParameters^.OffsetKPickPack;
			ELSE
				Lunghezza := Dimensioni_Pinza.Lunghezza;
			END_IF
		ELSIF  Mission^.JPickLT = 1 AND  Mission^.JPickVO = 1 THEN	// se trasversale ( PARALLELO A Y) e in orrizzontale
			Larghezza :=  Mission^.XDim;
			IF Mission^.YDim + PickPlaceParameters^.OffsetKPickPack >= Dimensioni_Pinza.Lunghezza THEN
				Lunghezza := ModuleAX_K^.Ax^.Status.ActPosition;
			ELSE
				Lunghezza := Dimensioni_Pinza.Lunghezza;
			END_IF
		ELSE
			Larghezza := Dimensioni_Pinza.Larghezza;
			Lunghezza := ModuleAX_K^.AxisPar^.MaxPosition;
		END_IF
		
	WAMANAGER_CICLO_DEPOSITO_PACCO_RUN:
		IF Mission^.JPickLT = 0 AND Mission^.JPickVO = 0 THEN // se longitudinale ( PARALLELO A X) e in verticale
			Larghezza :=  Mission^.ZDim;
			IF Mission^.XDim + PickPlaceParameters^.OffsetKPickPack >= Dimensioni_Pinza.Lunghezza THEN
				Lunghezza := Mission^.XDim + PickPlaceParameters^.OffsetKPickPack;
			ELSE
				Lunghezza := Dimensioni_Pinza.Lunghezza;
			END_IF
		ELSIF  Mission^.JPickLT = 0 AND  Mission^.JPickVO = 1 THEN	// se longitudinale ( PARALLELO A X) e in orrizzontale
			Larghezza :=  Mission^.YDim;
			IF Mission^.XDim + PickPlaceParameters^.OffsetKPickPack >= Dimensioni_Pinza.Lunghezza THEN
				Lunghezza := Mission^.XDim + PickPlaceParameters^.OffsetKPickPack;
			ELSE
				Lunghezza := Dimensioni_Pinza.Lunghezza;
			END_IF
		ELSIF  Mission^.JPickLT = 1 AND  Mission^.JPickVO = 0 THEN	// se trasversale ( PARALLELO A Y) e in verticale
			Larghezza :=  Mission^.XDim;
			IF Mission^.ZDim + PickPlaceParameters^.OffsetKPickPack >= Dimensioni_Pinza.Lunghezza THEN
				Lunghezza := Mission^.ZDim + PickPlaceParameters^.OffsetKPickPack;
			ELSE
				Lunghezza := Dimensioni_Pinza.Lunghezza;
			END_IF
		ELSIF  Mission^.JPickLT = 1 AND  Mission^.JPickVO = 1 THEN	// se trasversale ( PARALLELO A Y) e in orrizzontale
			Larghezza :=  Mission^.XDim;
			IF Mission^.YDim + PickPlaceParameters^.OffsetKPickPack >= Dimensioni_Pinza.Lunghezza THEN
				Lunghezza := ModuleAX_K^.Ax^.Status.ActPosition;
			ELSE
				Lunghezza := Dimensioni_Pinza.Lunghezza;
			END_IF
		ELSE
			Larghezza := Dimensioni_Pinza.Larghezza;
			Lunghezza := ModuleAX_K^.AxisPar^.MaxPosition;
		END_IF
					
END_CASE
(************************************ Ingombri Pinza ******************************************)

(* Valuto l' ingombro superficiale massimo *)
IngombroSuperficialePinzaMAX := SQRT((Larghezza * Larghezza) + (Lunghezza * Lunghezza));

(* Valuto l' ingombro Verticale massimo *)
IngombroVerticalePinzaMAX := Dimensione_Z_ElementoInPresaX_Ingombro;

(* Ingombro ottimizzato della pinza REAL-TIME *)
IngombroOttimizzatoX := ABS(IngombroSuperficialePinzaMAX * SIN(deg_to_rad((ATAN(Larghezza/Lunghezza)*1/0.017+ ModuleAX_J^.Ax^.AxRef^.NcToPlc.ActPos))));
IngombroOttimizzatoY := ABS(IngombroSuperficialePinzaMAX * COS(deg_to_rad((ATAN(Larghezza/Lunghezza)*1/0.017+ ModuleAX_J^.Ax^.AxRef^.NcToPlc.ActPos))));

(* Abilitazione dell'uso degli ingombri ottimizzati *)
IF AbilitaCalcoloIngombroOttimizzato THEN
	IngombroX := IngombroOttimizzatoX;
	IngombroY := IngombroOttimizzatoY;
ELSE
	IngombroX := IngombroSuperficialePinzaMAX;
	IngombroY := IngombroSuperficialePinzaMAX;
END_IF

IngombroSuperficialePinzaMAX_Global := IngombroSuperficialePinzaMAX;
IngombroXPinzaOttimizzato_Global 	:= IngombroX;
IngombroYPinzaOttimizzato_Global 	:= IngombroY;
(**********************************************************************************************)
(**********************************************************************************************)

(* Quota di Fuori-Ingombro della X rispetto le colonne, valutando l'ingombro effettivo della pinza *)
IF ModuleAX_X^.Ax^.AxRef^.Status.PositiveDirection THEN //Direzione POSITIVA 
	IF (ModuleAX_X^.Ax^.Status.ActPosition - IngombroX/ 2)-50 >= (WorkFootprint^[6].X + WorkFootprint^[6].XDim) THEN
		QuotaX_ConsensoRotazionePinza_RaggiuntaTMP := TRUE;
	ELSE
		QuotaX_ConsensoRotazionePinza_RaggiuntaTMP := FALSE;
	END_IF
ELSIF ModuleAX_X^.Ax^.AxRef^.Status.NegativeDirection (*OR WorkArea^[Mission^.PPick].X >= WorkArea^[Mission^.PPlace].X*) THEN //Direzione NEGATIVA 
	IF (ModuleAX_X^.Ax^.Status.ActPosition + IngombroX/ 2)+50 >(WorkFootprint^[6].X)(* OR WorkArea^[Mission^.PPick].X >= WorkArea^[Mission^.PPlace].X *)THEN
		QuotaX_ConsensoRotazionePinza_RaggiuntaTMP := TRUE;
	ELSE
		QuotaX_ConsensoRotazionePinza_RaggiuntaTMP := FALSE;
	END_IF
ELSIF WorkAreaManager^.State = WAMANAGER_CICLO_PRELIEVO_PACCO_RUN AND Mission^.TPick = TPICK_PACK AND (ModuleAX_X^.Ax^.AxRef^.NcToPlc.ActPos >= WorkPickPoint^[Mission^.PPick].Xh - 10 AND ModuleAX_X^.Ax^.AxRef^.NcToPlc.ActPos <= WorkPickPoint^[Mission^.PPick].Xh +10) THEN
	ConsensoTraslazioneY_TraColonneTMP := TRUE;
ELSE 
	QuotaX_ConsensoRotazionePinza_RaggiuntaTMP := FALSE;
END_IF

CASE WorkAreaManager^.State OF
	WAMANAGER_NOP: 
		CalcolaIngombro := TRUE;
	
	WAMANAGER_CICLO_RIPOSO_INIT: 
		CalcolaIngombro := TRUE;
		
	WAMANAGER_CICLO_RIPOSO_RUN:
		IF CalcolaIngombro THEN
			CalcolaIngombro := FALSE;
			(* Definisco il tipo di area in cui si trova a lavorare il pallettizzatore *)
			AreaInLavoroPositiva := FALSE;
			AreaInLavoroNegativa := FALSE;
			AreaInLavoroPositivaNegativa := TRUE; 
			
			(**************************************************************************************************************************************************)
			(* Ingombro ottimizzato della pinza sul punto di prelievo *)
			(**************************************************************************************************************************************************)
			IngombroOttimizzatoX_InPuntoDiPrelievo := ABS(IngombroSuperficialePinzaMAX * SIN(deg_to_rad((ATAN(Larghezza/Lunghezza)*1/0.017+ Mission^.JPick))));
			IngombroOttimizzatoY_InPuntoDiPrelievo := ABS(IngombroSuperficialePinzaMAX * COS(deg_to_rad((ATAN(Larghezza/Lunghezza)*1/0.017+ Mission^.JPick))));
			(**************************************************************************************************************************************************)
			(* Ingombro ottimizzato della pinza sul punto di deposito *)
			(**************************************************************************************************************************************************)
			IngombroOttimizzatoX_InPuntoDiDeposito := ABS(IngombroSuperficialePinzaMAX * SIN(deg_to_rad((ATAN(Larghezza/Lunghezza)*1/0.017+ Mission^.JPlace))));
			IngombroOttimizzatoY_InPuntoDiDeposito := ABS(IngombroSuperficialePinzaMAX * COS(deg_to_rad((ATAN(Larghezza/Lunghezza)*1/0.017+ Mission^.JPlace))));
						
			(**************************************************************************************************************************************************)
			(**************************************************************************************************************************************************)
						
			(* Valuto la direzione della X *)
			DirezioneXPositiva := TFDirezioneAssePositiva(Posizione_Attuale:=ModuleAX_X^.Ax^.Status.ActPosition,Posizione_Finale:=Mission^.XPick);
			DirezioneXNegativa := NOT DirezioneXPositiva;
				
			(* Valuto se gli assi sono in finestra di prelievo *)
			AsseXInFinestraDiRiposo := TFAsseInFinestra(Posizione_Attuale:=ModuleAx_X^.Ax^.AxRef^.NcToPlc.ActPos,Posizione_Finale:=Mission^.XPick,FinestraDiControllo:=10);
			AsseYInFinestraDiRiposo := TFAsseInFinestra(Posizione_Attuale:=ModuleAx_Y^.Ax^.AxRef^.NcToPlc.ActPos,Posizione_Finale:=Mission^.YPick,FinestraDiControllo:=10);
			AsseJInFinestraDiRiposo := TFAsseInFinestra(Posizione_Attuale:=ModuleAx_J^.Ax^.AxRef^.NcToPlc.ActPos,Posizione_Finale:=Mission^.JPick,FinestraDiControllo:=5);
			(* Valuto se gli assi sono in finestra di destinazione *)
			AsseXInFinestraDiDestinazione := TFAsseInFinestra(Posizione_Attuale:=ModuleAx_X^.Ax^.AxRef^.NcToPlc.ActPos,Posizione_Finale:=Mission^.XPick,FinestraDiControllo:=10);
			AsseYInFinestraDiDestinazione := TFAsseInFinestra(Posizione_Attuale:=ModuleAx_Y^.Ax^.AxRef^.NcToPlc.ActPos,Posizione_Finale:=Mission^.YPick,FinestraDiControllo:=10);
			AsseJInFinestraDiDestinazione := TFAsseInFinestra(Posizione_Attuale:=ModuleAx_J^.Ax^.AxRef^.NcToPlc.ActPos,Posizione_Finale:=Mission^.JPick,FinestraDiControllo:=5);
			
			(**************************************************************************************************************************************************)
			(* Ingombro MASSIMO della pinza durante il transito *)
			(**************************************************************************************************************************************************)
			//Calcolo ingombro attuale
			IngombroOttimizzatoX_InTransito := ABS(IngombroSuperficialePinzaMAX * SIN(deg_to_rad((ATAN(Larghezza/Lunghezza)*1/0.017+ ModuleAx_J^.Ax^.AxRef^.NcToPlc.ActPos)))); //Ingombro Attuale direzione X
			IngombroOttimizzatoY_InTransito := ABS(IngombroSuperficialePinzaMAX * COS(deg_to_rad((ATAN(Larghezza/Lunghezza)*1/0.017+ ModuleAx_J^.Ax^.AxRef^.NcToPlc.ActPos)))); //Ingombro Attuale direzione Y		
			IF NOT AsseJInFinestraDiDestinazione THEN
				IF REAL_TO_INT(ModuleAx_J^.Ax^.AxRef^.NcToPlc.ActPos) <= REAL_TO_INT(Mission^.JPick) THEN //Se l'angolo attuale di rotazione della pinza è INFERIORE alla posizione di destinazione
					FOR Angolo := REAL_TO_INT(ModuleAx_J^.Ax^.AxRef^.NcToPlc.ActPos) TO REAL_TO_INT(Mission^.JPick) DO //Valuto tutti i gradi di rotazione in direzione CRESCENTE fino all'angolo di destinazione
						IF IngombroOttimizzatoX_InTransito < ABS(IngombroSuperficialePinzaMAX * SIN(deg_to_rad((ATAN(Larghezza/Lunghezza)*1/0.017+ Angolo)))) THEN
							IngombroOttimizzatoX_InTransito := ABS(IngombroSuperficialePinzaMAX * SIN(deg_to_rad((ATAN(Larghezza/Lunghezza)*1/0.017+ Angolo)))) ;
						END_IF
						IF IngombroOttimizzatoY_InTransito < ABS(IngombroSuperficialePinzaMAX * COS(deg_to_rad((ATAN(Larghezza/Lunghezza)*1/0.017+ Angolo)))) THEN
							IngombroOttimizzatoY_InTransito := ABS(IngombroSuperficialePinzaMAX * COS(deg_to_rad((ATAN(Larghezza/Lunghezza)*1/0.017+ Angolo))));
						END_IF
					END_FOR
				ELSIF REAL_TO_INT(ModuleAx_J^.Ax^.AxRef^.NcToPlc.ActPos) >= REAL_TO_INT(Mission^.JPick) THEN //Se l'angolo attuale di rotazione della pinza è MAGGIORE alla posizione di destinazione
					FOR Angolo := REAL_TO_INT(ModuleAx_J^.Ax^.AxRef^.NcToPlc.ActPos) TO REAL_TO_INT(Mission^.JPick) BY -1 DO //Valuto tutti i gradi di rotazione in direzione DECRESCENTE fino all'angolo di destinazione
						IF IngombroOttimizzatoX_InTransito < ABS(IngombroSuperficialePinzaMAX * SIN(deg_to_rad((ATAN(Larghezza/Lunghezza)*1/0.017+ Angolo)))) THEN
							IngombroOttimizzatoX_InTransito := ABS(IngombroSuperficialePinzaMAX * SIN(deg_to_rad((ATAN(Larghezza/Lunghezza)*1/0.017+ Angolo)))) ;
						END_IF
						IF IngombroOttimizzatoY_InTransito < ABS(IngombroSuperficialePinzaMAX * COS(deg_to_rad((ATAN(Larghezza/Lunghezza)*1/0.017+ Angolo)))) THEN
							IngombroOttimizzatoY_InTransito := ABS(IngombroSuperficialePinzaMAX * COS(deg_to_rad((ATAN(Larghezza/Lunghezza)*1/0.017+ Angolo))));
						END_IF
					END_FOR
				END_IF
			END_IF
		
			(* Valutazione colonne in base al verso del pallettizzatore: verso stabilito guardando il pallettizzatore con la linea alle spalle *)
			CASE VERSO_PALLETTIZZATORE OF
				PALLETTIZZATORE_DX:	// Colonna 6:DX, 5:SX
					(* Valuto la posizione attuale *)
					IF (ModuleAX_Y^.Ax^.Status.ActPosition - IngombroY/2 - OffsetSicurezza_Y <= WorkFootprint^[6].Y) THEN //Posizione Pinza - Metà ingombro - Offset sicurezza <= Ingombro colonna DX
						QuotaFuoriIngombro_Attuale_Y := WorkFootprint^[6].Y + IngombroY/2 + OffsetSicurezza_Y;
						Pinza_InIngombroColonne_Attuale := TRUE;
					ELSIF (ModuleAX_Y^.Ax^.Status.ActPosition + IngombroY/2 + OffsetSicurezza_Y >= WorkFootprint^[5].Y) THEN //Posizione Pinza + Metà ingombro + Offset sicurezza >= Ingombro colonna SX
						QuotaFuoriIngombro_Attuale_Y := WorkFootprint^[5].Y - IngombroY/2 - OffsetSicurezza_Y;
						Pinza_InIngombroColonne_Attuale := TRUE;
					ELSE
						QuotaFuoriIngombro_Attuale_Y := ModuleAX_Y^.Ax^.Status.ActPosition;
						Pinza_InIngombroColonne_Attuale := FALSE;
					END_IF
					
					(* Valuto la posizione futura - Missione di prelievo *)
					IF (Mission^.YPick - IngombroOttimizzatoY_InPuntoDiPrelievo/2 - OffsetSicurezza_Y <= WorkFootprint^[6].Y) THEN //Posizione Pinza - Metà ingombro - Offset sicurezza <= Ingombro colonna DX
						QuotaFuoriIngombro_Prelievo_Y := WorkFootprint^[6].Y + IngombroOttimizzatoY_InPuntoDiPrelievo/2 + OffsetSicurezza_Y; 
						Pinza_InIngombroColonne_Destinazione := TRUE;
					ELSIF (Mission^.YPick + IngombroOttimizzatoY_InPuntoDiPrelievo/2 + OffsetSicurezza_Y >= WorkFootprint^[5].Y) THEN //Posizione Pinza + Metà ingombro + Offset sicurezza >= Ingombro colonna SX
						QuotaFuoriIngombro_Prelievo_Y := WorkFootprint^[5].Y - IngombroOttimizzatoY_InPuntoDiPrelievo/2 - OffsetSicurezza_Y;
						Pinza_InIngombroColonne_Destinazione := TRUE;
					ELSE
						QuotaFuoriIngombro_Prelievo_Y := Mission^.YPick;
						Pinza_InIngombroColonne_Destinazione := FALSE;
					END_IF
					
					(* Valuto la posizione futura - Missione di Deposito *)
					IF (Mission^.YPlace - IngombroOttimizzatoY_InPuntoDiDeposito/2 - OffsetSicurezza_Y <= WorkFootprint^[6].Y) THEN //Posizione Pinza - Metà ingombro - Offset sicurezza <= Ingombro colonna DX
						QuotaFuoriIngombro_Deposito_Y := WorkFootprint^[6].Y + IngombroOttimizzatoY_InPuntoDiPrelievo/2 + OffsetSicurezza_Y;
						Pinza_InIngombroColonne_Destinazione := TRUE;
					ELSIF (Mission^.YPlace + IngombroOttimizzatoY_InPuntoDiDeposito/2 + OffsetSicurezza_Y >= WorkFootprint^[5].Y) THEN //Posizione Pinza + Metà ingombro + Offset sicurezza >= Ingombro colonna SX
						QuotaFuoriIngombro_Deposito_Y := WorkFootprint^[5].Y - IngombroOttimizzatoY_InPuntoDiPrelievo/2 - OffsetSicurezza_Y;
						Pinza_InIngombroColonne_Destinazione := TRUE;
					ELSE
						QuotaFuoriIngombro_Deposito_Y := Mission^.YPlace;
						Pinza_InIngombroColonne_Destinazione := FALSE;
					END_IF
					
					(* Valuto la posizione attuale Y e la posizione di destinazione Y e l'ingombro massimo che posso avere durante il transito *)
					IF (Mission^.YPick - IngombroOttimizzatoY_InTransito/2 - OffsetSicurezza_Y <= WorkFootprint^[6].Y) THEN //Posizione Pinza - Metà ingombro - Offset sicurezza <= Ingombro colonna DX
						Pinza_InIngombroColonne_Transito := TRUE;
					ELSIF (Mission^.YPick + IngombroOttimizzatoY_InTransito/2 + OffsetSicurezza_Y >= WorkFootprint^[5].Y) THEN //Posizione Pinza + Metà ingombro + Offset sicurezza >= Ingombro colonna SX
						Pinza_InIngombroColonne_Transito := TRUE;
					ELSE
						Pinza_InIngombroColonne_Transito := FALSE;
					END_IF
						
				PALLETTIZZATORE_SX: // Colonna 6:SX, 5:DX
					(* Valuto la posizione attuale *)
					IF (ModuleAX_Y^.Ax^.Status.ActPosition - IngombroY/2 - OffsetSicurezza_Y <= WorkFootprint^[5].Y) THEN //Posizione Pinza - Metà ingombro - Offset sicurezza <= Ingombro colonna 
						Pinza_InIngombroColonne_Attuale := TRUE;
					ELSIF (ModuleAX_Y^.Ax^.Status.ActPosition + IngombroY/2 + OffsetSicurezza_Y >= WorkFootprint^[6].Y) THEN //Posizione Pinza + Metà ingombro + Offset sicurezza <= Ingombro colonna 
						Pinza_InIngombroColonne_Attuale := TRUE;
					ELSE
						Pinza_InIngombroColonne_Attuale := FALSE;
					END_IF
					(* Valuto la posizione futura - Missione di prelievo *)
					IF (Mission^.YPick - IngombroOttimizzatoX_InPuntoDiPrelievo/2 - OffsetSicurezza_Y <= WorkFootprint^[5].Y) THEN //Posizione Pinza - Metà ingombro - Offset sicurezza <= Ingombro colonna 
						Pinza_InIngombroColonne_Destinazione := TRUE;
					ELSIF (Mission^.YPick + IngombroOttimizzatoX_InPuntoDiPrelievo/2 + OffsetSicurezza_Y >= WorkFootprint^[6].Y) THEN //Posizione Pinza + Metà ingombro + Offset sicurezza <= Ingombro colonna 
						Pinza_InIngombroColonne_Destinazione := TRUE;
					ELSE
						Pinza_InIngombroColonne_Destinazione := FALSE;
					END_IF
					
					(* Valuto la posizione futura - Missione di Deposito *)
					IF (Mission^.YPick - IngombroOttimizzatoX_InPuntoDiDeposito/2 - OffsetSicurezza_Y <= WorkFootprint^[5].Y) THEN //Posizione Pinza - Metà ingombro - Offset sicurezza <= Ingombro colonna 
						Pinza_InIngombroColonne_Destinazione := TRUE;
					ELSIF (Mission^.YPick + IngombroOttimizzatoX_InPuntoDiDeposito/2 + OffsetSicurezza_Y >= WorkFootprint^[6].Y) THEN //Posizione Pinza + Metà ingombro + Offset sicurezza <= Ingombro colonna 
						Pinza_InIngombroColonne_Destinazione := TRUE;
					ELSE
						Pinza_InIngombroColonne_Destinazione := FALSE;
					END_IF
					
					(* Valuto la posizione attuale Y e la posizione di destinazione Y e l'ingombro massimo che posso avere durante il transito *)
					IF (Mission^.YPick - IngombroOttimizzatoY_InTransito/2 - OffsetSicurezza_Y <= WorkFootprint^[5].Y) THEN //Posizione Pinza - Metà ingombro - Offset sicurezza <= Ingombro colonna 
						Pinza_InIngombroColonne_Transito := TRUE;
					ELSIF (Mission^.YPick + IngombroOttimizzatoY_InTransito/2 + OffsetSicurezza_Y >= WorkFootprint^[6].Y) THEN //Posizione Pinza + Metà ingombro + Offset sicurezza <= Ingombro colonna 
						Pinza_InIngombroColonne_Transito := TRUE;
					ELSE
						Pinza_InIngombroColonne_Transito := FALSE;
					END_IF
			END_CASE		
			(* Se sono in ingombro nella posizione attuale o nella posizione di destinazione, devo andare fuori-ingombro con la Y *)
			IF (Pinza_InIngombroColonne_Attuale OR Pinza_InIngombroColonne_Destinazione OR Pinza_InIngombroColonne_Transito) THEN 
				IF (AsseXInFinestraDiRiposo AND AsseYInFinestraDiRiposo AND AsseJInFinestraDiRiposo) THEN //Se sono in finestra di riposo con tutti gli assi non devo andare fuori-ingombro con la Y
					FuoriIngombroYNecessarioTMP := FALSE;
				ELSE
					FuoriIngombroYNecessarioTMP := TRUE;
				END_IF
			ELSE
				FuoriIngombroYNecessarioTMP := FALSE;
			END_IF
		END_IF
								
	WAMANAGER_CICLO_RIPOSO_END: 
		CalcolaIngombro := TRUE;
			
	WAMANAGER_CICLO_PALL_INIT:
		CalcolaIngombro := TRUE;
	
	WAMANAGER_CICLO_PRELIEVO_PALL_RUN:
		IF CalcolaIngombro THEN
			CalcolaIngombro := FALSE;
			(* Definisco il tipo di area in cui si trova a lavorare il pallettizzatore *)
			AreaInLavoroPositiva := FALSE;
			AreaInLavoroNegativa := FALSE;
			AreaInLavoroPositivaNegativa := FALSE; 
			IF WorkArea^[Mission^.PPick].X >= (WorkFootprint^[5].X + WorkFootprint^[5].XDim) AND 	//se la piazzola di prelievo ha quota maggiore rispetto le colonne centrali
				ModuleAx_X^.Ax^.AxRef^.NcToPlc.ActPos >= (WorkFootprint^[5].X + WorkFootprint^[5].XDim)  THEN //Sono già nella campata positiva
					AreaInLavoroPositiva := TRUE;
			ELSIF WorkArea^[Mission^.PPick].X <= WorkFootprint^[5].X AND 	//se la piazzola di prelievo ha quota maggiore della piazzola di deposito e
				ModuleAx_X^.Ax^.AxRef^.NcToPlc.ActPos <= WorkFootprint^[5].X  THEN //Sono già nella campata negativa
					AreaInLavoroNegativa := TRUE;
			ELSE
				AreaInLavoroPositiva := FALSE;
				AreaInLavoroNegativa := FALSE;
				AreaInLavoroPositivaNegativa := TRUE;
			END_IF
			
			(**************************************************************************************************************************************************)
			(* Ingombro ottimizzato della pinza sul punto di prelievo *)
			(**************************************************************************************************************************************************)
			IngombroOttimizzatoX_InPuntoDiPrelievo := ABS(IngombroSuperficialePinzaMAX * SIN(deg_to_rad((ATAN(Larghezza/Lunghezza)*1/0.017+ Mission^.JPick))));
			IngombroOttimizzatoY_InPuntoDiPrelievo := ABS(IngombroSuperficialePinzaMAX * COS(deg_to_rad((ATAN(Larghezza/Lunghezza)*1/0.017+ Mission^.JPick))));
			(**************************************************************************************************************************************************)
			(* Ingombro ottimizzato della pinza sul punto di deposito *)
			(**************************************************************************************************************************************************)
			IngombroOttimizzatoX_InPuntoDiDeposito := ABS(IngombroSuperficialePinzaMAX * SIN(deg_to_rad((ATAN(Larghezza/Lunghezza)*1/0.017+ Mission^.JPlace))));
			IngombroOttimizzatoY_InPuntoDiDeposito := ABS(IngombroSuperficialePinzaMAX * COS(deg_to_rad((ATAN(Larghezza/Lunghezza)*1/0.017+ Mission^.JPlace))));
						
			(**************************************************************************************************************************************************)
			(**************************************************************************************************************************************************)
						
			(* Valuto la direzione della X *)
			DirezioneXPositiva := TFDirezioneAssePositiva(Posizione_Attuale:=ModuleAX_X^.Ax^.Status.ActPosition,Posizione_Finale:=Mission^.XPick);
			DirezioneXNegativa := NOT DirezioneXPositiva;
				
			(* Valuto se gli assi sono in finestra di destinazione *)
			AsseXInFinestraDiDestinazione := TFAsseInFinestra(Posizione_Attuale:=ModuleAx_X^.Ax^.AxRef^.NcToPlc.ActPos,Posizione_Finale:=Mission^.XPick,FinestraDiControllo:=10);
			AsseYInFinestraDiDestinazione := TFAsseInFinestra(Posizione_Attuale:=ModuleAx_Y^.Ax^.AxRef^.NcToPlc.ActPos,Posizione_Finale:=Mission^.YPick,FinestraDiControllo:=10);
			AsseJInFinestraDiDestinazione := TFAsseInFinestra(Posizione_Attuale:=ModuleAx_J^.Ax^.AxRef^.NcToPlc.ActPos,Posizione_Finale:=Mission^.JPick,FinestraDiControllo:=5);
			
			(**************************************************************************************************************************************************)
			(* Ingombro MASSIMO della pinza durante il transito *)
			(**************************************************************************************************************************************************)
			//Calcolo ingombro attuale
			IngombroOttimizzatoX_InTransito := ABS(IngombroSuperficialePinzaMAX * SIN(deg_to_rad((ATAN(Larghezza/Lunghezza)*1/0.017+ ModuleAx_J^.Ax^.AxRef^.NcToPlc.ActPos)))); //Ingombro Attuale direzione X
			IngombroOttimizzatoY_InTransito := ABS(IngombroSuperficialePinzaMAX * COS(deg_to_rad((ATAN(Larghezza/Lunghezza)*1/0.017+ ModuleAx_J^.Ax^.AxRef^.NcToPlc.ActPos)))); //Ingombro Attuale direzione Y		
			IF NOT AsseJInFinestraDiDestinazione THEN
				IF REAL_TO_INT(ModuleAx_J^.Ax^.AxRef^.NcToPlc.ActPos) <= REAL_TO_INT(Mission^.JPick) THEN
					FOR Angolo := REAL_TO_INT(ModuleAx_J^.Ax^.AxRef^.NcToPlc.ActPos) TO REAL_TO_INT(Mission^.JPick)  DO
						IF IngombroOttimizzatoX_InTransito < ABS(IngombroSuperficialePinzaMAX * SIN(deg_to_rad((ATAN(Larghezza/Lunghezza)*1/0.017+ Angolo)))) THEN
							IngombroOttimizzatoX_InTransito := ABS(IngombroSuperficialePinzaMAX * SIN(deg_to_rad((ATAN(Larghezza/Lunghezza)*1/0.017+ Angolo)))) ;
						END_IF
						IF IngombroOttimizzatoY_InTransito < ABS(IngombroSuperficialePinzaMAX * COS(deg_to_rad((ATAN(Larghezza/Lunghezza)*1/0.017+ Angolo)))) THEN
							IngombroOttimizzatoY_InTransito := ABS(IngombroSuperficialePinzaMAX * COS(deg_to_rad((ATAN(Larghezza/Lunghezza)*1/0.017+ Angolo))));
						END_IF
					END_FOR
				END_IF
			END_IF
		
			(* Valutazione colonne in base al verso del pallettizzatore *)
			CASE VERSO_PALLETTIZZATORE OF
				PALLETTIZZATORE_DX:	// Colonna 6:DX, 5:SX
					(* Valuto la posizione attuale *)
					IF (ModuleAX_Y^.Ax^.Status.ActPosition - IngombroY/2 - OffsetSicurezza_Y <= WorkFootprint^[6].Y) OR //Posizione Pinza - Metà ingombro - Offset sicurezza <= Ingombro colonna 
						(ModuleAX_Y^.Ax^.Status.ActPosition + IngombroY/2 + OffsetSicurezza_Y >= WorkFootprint^[5].Y) THEN //Posizione Pinza - Metà ingombro - Offset sicurezza <= Ingombro colonna 
							Pinza_InIngombroColonne_Attuale := TRUE;
					ELSE
							Pinza_InIngombroColonne_Attuale := FALSE;
					END_IF
					(* Valuto la posizione futura - Missione di prelievo *)
					IF (Mission^.YPick - IngombroOttimizzatoX_InPuntoDiPrelievo/2 - OffsetSicurezza_Y <= WorkFootprint^[6].Y) OR //Posizione Pinza - Metà ingombro - Offset sicurezza <= Ingombro colonna 
						(Mission^.YPick + IngombroOttimizzatoX_InPuntoDiPrelievo/2 + OffsetSicurezza_Y >= WorkFootprint^[5].Y) THEN //Posizione Pinza - Metà ingombro - Offset sicurezza <= Ingombro colonna 
							Pinza_InIngombroColonne_Destinazione := TRUE;
					ELSE
							Pinza_InIngombroColonne_Destinazione := FALSE;
					END_IF
					
					(* Valuto la posizione futura - Missione di Deposito *)
					IF (Mission^.YPick - IngombroOttimizzatoX_InPuntoDiDeposito/2 - OffsetSicurezza_Y <= WorkFootprint^[6].Y) OR //Posizione Pinza - Metà ingombro - Offset sicurezza <= Ingombro colonna 
						(Mission^.YPick + IngombroOttimizzatoX_InPuntoDiDeposito/2 + OffsetSicurezza_Y >= WorkFootprint^[5].Y) THEN //Posizione Pinza - Metà ingombro - Offset sicurezza <= Ingombro colonna 
							Pinza_InIngombroColonne_Destinazione := TRUE;
					ELSE
							Pinza_InIngombroColonne_Destinazione := FALSE;
					END_IF
					
					(* Valuto la posizione attuale Y e la posizione di destinazione Y e l'ingombro massimo che posso avere durante il transito *)
					IF (Mission^.YPick - IngombroOttimizzatoY_InTransito/2 - OffsetSicurezza_Y <= WorkFootprint^[6].Y) OR //Posizione Pinza - Metà ingombro - Offset sicurezza <= Ingombro colonna 
						(Mission^.YPick + IngombroOttimizzatoY_InTransito/2 + OffsetSicurezza_Y >= WorkFootprint^[5].Y) THEN //Posizione Pinza - Metà ingombro - Offset sicurezza <= Ingombro colonna 
							Pinza_InIngombroColonne_Transito := TRUE;
					ELSE
							Pinza_InIngombroColonne_Transito := FALSE;
					END_IF
						
				PALLETTIZZATORE_SX: // Colonna 6:SX, 5:DX
					(* Valuto la posizione attuale *)
					IF (ModuleAX_Y^.Ax^.Status.ActPosition - IngombroY/2 - OffsetSicurezza_Y <= WorkFootprint^[5].Y) OR //Posizione Pinza - Metà ingombro - Offset sicurezza <= Ingombro colonna 
						(ModuleAX_Y^.Ax^.Status.ActPosition + IngombroY/2 + OffsetSicurezza_Y >= WorkFootprint^[6].Y) THEN //Posizione Pinza - Metà ingombro - Offset sicurezza <= Ingombro colonna 
							Pinza_InIngombroColonne_Attuale := TRUE;
					ELSE
							Pinza_InIngombroColonne_Attuale := FALSE;
					END_IF
					(* Valuto la posizione futura - Missione di prelievo *)
					IF (Mission^.YPick - IngombroOttimizzatoX_InPuntoDiPrelievo/2 - OffsetSicurezza_Y <= WorkFootprint^[5].Y) OR //Posizione Pinza - Metà ingombro - Offset sicurezza <= Ingombro colonna 
						(Mission^.YPick + IngombroOttimizzatoX_InPuntoDiPrelievo/2 + OffsetSicurezza_Y >= WorkFootprint^[6].Y) THEN //Posizione Pinza - Metà ingombro - Offset sicurezza <= Ingombro colonna 
							Pinza_InIngombroColonne_Destinazione := TRUE;
					ELSE
							Pinza_InIngombroColonne_Destinazione := FALSE;
					END_IF
					
					(* Valuto la posizione futura - Missione di Deposito *)
					IF (Mission^.YPick - IngombroOttimizzatoX_InPuntoDiDeposito/2 - OffsetSicurezza_Y <= WorkFootprint^[5].Y) OR //Posizione Pinza - Metà ingombro - Offset sicurezza <= Ingombro colonna 
						(Mission^.YPick + IngombroOttimizzatoX_InPuntoDiDeposito/2 + OffsetSicurezza_Y >= WorkFootprint^[6].Y) THEN //Posizione Pinza - Metà ingombro - Offset sicurezza <= Ingombro colonna 
							Pinza_InIngombroColonne_Destinazione := TRUE;
					ELSE
							Pinza_InIngombroColonne_Destinazione := FALSE;
					END_IF
					
					(* Valuto la posizione attuale Y e la posizione di destinazione Y e l'ingombro massimo che posso avere durante il transito *)
					IF (Mission^.YPick - IngombroOttimizzatoY_InTransito/2 - OffsetSicurezza_Y <= WorkFootprint^[5].Y) OR //Posizione Pinza - Metà ingombro - Offset sicurezza <= Ingombro colonna 
						(Mission^.YPick + IngombroOttimizzatoY_InTransito/2 + OffsetSicurezza_Y >= WorkFootprint^[6].Y) THEN //Posizione Pinza - Metà ingombro - Offset sicurezza <= Ingombro colonna 
							Pinza_InIngombroColonne_Transito := TRUE;
					ELSE
							Pinza_InIngombroColonne_Transito := FALSE;
					END_IF
			END_CASE		
			(* Se sono in ingombro nella posizione attuale o nella posizione di destinazione, devo andare fuori-ingombro con la Y *)
			IF AreaInLavoroPositivaNegativa THEN
				FuoriIngombroYNecessarioTMP := TRUE;
			ELSE
				FuoriIngombroYNecessarioTMP := FALSE;
			END_IF
			
			IF (Pinza_InIngombroColonne_Attuale OR Pinza_InIngombroColonne_Destinazione OR Pinza_InIngombroColonne_Transito) THEN 
				FuoriIngombroYNecessarioTMP := TRUE;
			ELSE
				FuoriIngombroYNecessarioTMP := FALSE;
			END_IF
			
			IF (AsseXInFinestraDiDestinazione AND AsseYInFinestraDiDestinazione AND AsseJInFinestraDiDestinazione) THEN //Se sono in finestra di DESTINAZIONE con tutti gli assi non devo andare fuori-ingombro con la Y
				FuoriIngombroYNecessarioTMP := FALSE;
			ELSE
				FuoriIngombroYNecessarioTMP := TRUE;
			END_IF
			
			
		END_IF
		
	WAMANAGER_CICLO_PRELIEVO_PALL_END:
		CalcolaIngombro := TRUE;					
		
	WAMANAGER_CICLO_DEPOSITO_PALL_RUN:
		IF CalcolaIngombro THEN
			CalcolaIngombro := FALSE;
			(* Definisco il tipo di area in cui si trova a lavorare il pallettizzatore *)
			AreaInLavoroPositiva := FALSE;
			AreaInLavoroNegativa := FALSE;
			AreaInLavoroPositivaNegativa := FALSE; 
			IF ModuleAx_X^.Ax^.AxRef^.NcToPlc.ActPos >= (WorkFootprint^[5].X + WorkFootprint^[5].XDim) AND 	//se la piazzola di prelievo ha quota maggiore rispetto le colonne centrali
				WorkArea^[Mission^.PPlace].X >= (WorkFootprint^[5].X + WorkFootprint^[5].XDim)  THEN //la piazzola di deposito è nella campata positiva
					AreaInLavoroPositiva := TRUE;
			ELSIF ModuleAx_X^.Ax^.AxRef^.NcToPlc.ActPos <= WorkFootprint^[5].X AND 	//se la piazzola di prelievo ha quota maggiore della piazzola di deposito e
				WorkArea^[Mission^.PPlace].X <= WorkFootprint^[5].X  THEN //la piazzola di deposito è nella campata negativa
					AreaInLavoroNegativa := TRUE;
			ELSE
				AreaInLavoroPositiva := FALSE;
				AreaInLavoroNegativa := FALSE;
				AreaInLavoroPositivaNegativa := TRUE;
			END_IF
			
			(**************************************************************************************************************************************************)
			(* Ingombro ottimizzato della pinza sul punto di prelievo *)
			(**************************************************************************************************************************************************)
			IngombroOttimizzatoX_InPuntoDiPrelievo := ABS(IngombroSuperficialePinzaMAX * SIN(deg_to_rad((ATAN(Larghezza/Lunghezza)*1/0.017+ Mission^.JPick))));
			IngombroOttimizzatoY_InPuntoDiPrelievo := ABS(IngombroSuperficialePinzaMAX * COS(deg_to_rad((ATAN(Larghezza/Lunghezza)*1/0.017+ Mission^.JPick))));
			(**************************************************************************************************************************************************)
			(* Ingombro ottimizzato della pinza sul punto di deposito *)
			(**************************************************************************************************************************************************)
			IngombroOttimizzatoX_InPuntoDiDeposito := ABS(IngombroSuperficialePinzaMAX * SIN(deg_to_rad((ATAN(Larghezza/Lunghezza)*1/0.017+ Mission^.JPlace))));
			IngombroOttimizzatoY_InPuntoDiDeposito := ABS(IngombroSuperficialePinzaMAX * COS(deg_to_rad((ATAN(Larghezza/Lunghezza)*1/0.017+ Mission^.JPlace))));
						
			(**************************************************************************************************************************************************)
			(**************************************************************************************************************************************************)
						
			(* Valuto la direzione della X *)
			DirezioneXPositiva := TFDirezioneAssePositiva(Posizione_Attuale:=ModuleAX_X^.Ax^.Status.ActPosition,Posizione_Finale:=Mission^.XPick);
			DirezioneXNegativa := NOT DirezioneXPositiva;
				
			(* Valuto se gli assi sono in finestra di prelievo *)
			AsseXInFinestraDiRiposo := TFAsseInFinestra(Posizione_Attuale:=ModuleAx_X^.Ax^.AxRef^.NcToPlc.ActPos,Posizione_Finale:=Mission^.XPick,FinestraDiControllo:=10);
			AsseYInFinestraDiRiposo := TFAsseInFinestra(Posizione_Attuale:=ModuleAx_Y^.Ax^.AxRef^.NcToPlc.ActPos,Posizione_Finale:=Mission^.YPick,FinestraDiControllo:=10);
			AsseJInFinestraDiRiposo := TFAsseInFinestra(Posizione_Attuale:=ModuleAx_J^.Ax^.AxRef^.NcToPlc.ActPos,Posizione_Finale:=Mission^.JPick,FinestraDiControllo:=5);
			(* Valuto se gli assi sono in finestra di destinazione *)
			AsseXInFinestraDiDestinazione := TFAsseInFinestra(Posizione_Attuale:=ModuleAx_X^.Ax^.AxRef^.NcToPlc.ActPos,Posizione_Finale:=Mission^.XPick,FinestraDiControllo:=10);
			AsseYInFinestraDiDestinazione := TFAsseInFinestra(Posizione_Attuale:=ModuleAx_Y^.Ax^.AxRef^.NcToPlc.ActPos,Posizione_Finale:=Mission^.YPick,FinestraDiControllo:=10);
			AsseJInFinestraDiDestinazione := TFAsseInFinestra(Posizione_Attuale:=ModuleAx_J^.Ax^.AxRef^.NcToPlc.ActPos,Posizione_Finale:=Mission^.JPick,FinestraDiControllo:=5);
			
			(**************************************************************************************************************************************************)
			(* Ingombro MASSIMO della pinza durante il transito *)
			(**************************************************************************************************************************************************)
			//Calcolo ingombro attuale
			IngombroOttimizzatoX_InTransito := ABS(IngombroSuperficialePinzaMAX * SIN(deg_to_rad((ATAN(Larghezza/Lunghezza)*1/0.017+ ModuleAx_J^.Ax^.AxRef^.NcToPlc.ActPos)))); //Ingombro Attuale direzione X
			IngombroOttimizzatoY_InTransito := ABS(IngombroSuperficialePinzaMAX * COS(deg_to_rad((ATAN(Larghezza/Lunghezza)*1/0.017+ ModuleAx_J^.Ax^.AxRef^.NcToPlc.ActPos)))); //Ingombro Attuale direzione Y		
			IF NOT AsseJInFinestraDiDestinazione THEN
				IF REAL_TO_INT(ModuleAx_J^.Ax^.AxRef^.NcToPlc.ActPos) <= REAL_TO_INT(Mission^.JPick) THEN
					FOR Angolo := REAL_TO_INT(ModuleAx_J^.Ax^.AxRef^.NcToPlc.ActPos) TO REAL_TO_INT(Mission^.JPick)  DO
						IF IngombroOttimizzatoX_InTransito < ABS(IngombroSuperficialePinzaMAX * SIN(deg_to_rad((ATAN(Larghezza/Lunghezza)*1/0.017+ Angolo)))) THEN
							IngombroOttimizzatoX_InTransito := ABS(IngombroSuperficialePinzaMAX * SIN(deg_to_rad((ATAN(Larghezza/Lunghezza)*1/0.017+ Angolo)))) ;
						END_IF
						IF IngombroOttimizzatoY_InTransito < ABS(IngombroSuperficialePinzaMAX * COS(deg_to_rad((ATAN(Larghezza/Lunghezza)*1/0.017+ Angolo)))) THEN
							IngombroOttimizzatoY_InTransito := ABS(IngombroSuperficialePinzaMAX * COS(deg_to_rad((ATAN(Larghezza/Lunghezza)*1/0.017+ Angolo))));
						END_IF
					END_FOR
				END_IF
			END_IF
		
			(* Valutazione colonne in base al verso del pallettizzatore *)
			CASE VERSO_PALLETTIZZATORE OF
				PALLETTIZZATORE_DX:	// Colonna 6:DX, 5:SX
					(* Valuto la posizione attuale *)
					IF (ModuleAX_Y^.Ax^.Status.ActPosition - IngombroY/2 - OffsetSicurezza_Y <= WorkFootprint^[6].Y) OR //Posizione Pinza - Metà ingombro - Offset sicurezza <= Ingombro colonna 
						(ModuleAX_Y^.Ax^.Status.ActPosition + IngombroY/2 + OffsetSicurezza_Y >= WorkFootprint^[5].Y) THEN //Posizione Pinza - Metà ingombro - Offset sicurezza <= Ingombro colonna 
							Pinza_InIngombroColonne_Attuale := TRUE;
					ELSE
							Pinza_InIngombroColonne_Attuale := FALSE;
					END_IF
					(* Valuto la posizione futura - Missione di prelievo *)
					IF (Mission^.YPick - IngombroOttimizzatoX_InPuntoDiPrelievo/2 - OffsetSicurezza_Y <= WorkFootprint^[6].Y) OR //Posizione Pinza - Metà ingombro - Offset sicurezza <= Ingombro colonna 
						(Mission^.YPick + IngombroOttimizzatoX_InPuntoDiPrelievo/2 + OffsetSicurezza_Y >= WorkFootprint^[5].Y) THEN //Posizione Pinza - Metà ingombro - Offset sicurezza <= Ingombro colonna 
							Pinza_InIngombroColonne_Destinazione := TRUE;
					ELSE
							Pinza_InIngombroColonne_Destinazione := FALSE;
					END_IF
					
					(* Valuto la posizione futura - Missione di Deposito *)
					IF (Mission^.YPick - IngombroOttimizzatoX_InPuntoDiDeposito/2 - OffsetSicurezza_Y <= WorkFootprint^[6].Y) OR //Posizione Pinza - Metà ingombro - Offset sicurezza <= Ingombro colonna 
						(Mission^.YPick + IngombroOttimizzatoX_InPuntoDiDeposito/2 + OffsetSicurezza_Y >= WorkFootprint^[5].Y) THEN //Posizione Pinza - Metà ingombro - Offset sicurezza <= Ingombro colonna 
							Pinza_InIngombroColonne_Destinazione := TRUE;
					ELSE
							Pinza_InIngombroColonne_Destinazione := FALSE;
					END_IF
					
					(* Valuto la posizione attuale Y e la posizione di destinazione Y e l'ingombro massimo che posso avere durante il transito *)
					IF (Mission^.YPick - IngombroOttimizzatoY_InTransito/2 - OffsetSicurezza_Y <= WorkFootprint^[6].Y) OR //Posizione Pinza - Metà ingombro - Offset sicurezza <= Ingombro colonna 
						(Mission^.YPick + IngombroOttimizzatoY_InTransito/2 + OffsetSicurezza_Y >= WorkFootprint^[5].Y) THEN //Posizione Pinza - Metà ingombro - Offset sicurezza <= Ingombro colonna 
							Pinza_InIngombroColonne_Transito := TRUE;
					ELSE
							Pinza_InIngombroColonne_Transito := FALSE;
					END_IF
						
				PALLETTIZZATORE_SX: // Colonna 6:SX, 5:DX
					(* Valuto la posizione attuale *)
					IF (ModuleAX_Y^.Ax^.Status.ActPosition - IngombroY/2 - OffsetSicurezza_Y <= WorkFootprint^[5].Y) OR //Posizione Pinza - Metà ingombro - Offset sicurezza <= Ingombro colonna 
						(ModuleAX_Y^.Ax^.Status.ActPosition + IngombroY/2 + OffsetSicurezza_Y >= WorkFootprint^[6].Y) THEN //Posizione Pinza - Metà ingombro - Offset sicurezza <= Ingombro colonna 
							Pinza_InIngombroColonne_Attuale := TRUE;
					ELSE
							Pinza_InIngombroColonne_Attuale := FALSE;
					END_IF
					(* Valuto la posizione futura - Missione di prelievo *)
					IF (Mission^.YPick - IngombroOttimizzatoX_InPuntoDiPrelievo/2 - OffsetSicurezza_Y <= WorkFootprint^[5].Y) OR //Posizione Pinza - Metà ingombro - Offset sicurezza <= Ingombro colonna 
						(Mission^.YPick + IngombroOttimizzatoX_InPuntoDiPrelievo/2 + OffsetSicurezza_Y >= WorkFootprint^[6].Y) THEN //Posizione Pinza - Metà ingombro - Offset sicurezza <= Ingombro colonna 
							Pinza_InIngombroColonne_Destinazione := TRUE;
					ELSE
							Pinza_InIngombroColonne_Destinazione := FALSE;
					END_IF
					
					(* Valuto la posizione futura - Missione di Deposito *)
					IF (Mission^.YPick - IngombroOttimizzatoX_InPuntoDiDeposito/2 - OffsetSicurezza_Y <= WorkFootprint^[5].Y) OR //Posizione Pinza - Metà ingombro - Offset sicurezza <= Ingombro colonna 
						(Mission^.YPick + IngombroOttimizzatoX_InPuntoDiDeposito/2 + OffsetSicurezza_Y >= WorkFootprint^[6].Y) THEN //Posizione Pinza - Metà ingombro - Offset sicurezza <= Ingombro colonna 
							Pinza_InIngombroColonne_Destinazione := TRUE;
					ELSE
							Pinza_InIngombroColonne_Destinazione := FALSE;
					END_IF
					
					(* Valuto la posizione attuale Y e la posizione di destinazione Y e l'ingombro massimo che posso avere durante il transito *)
					IF (Mission^.YPick - IngombroOttimizzatoY_InTransito/2 - OffsetSicurezza_Y <= WorkFootprint^[5].Y) OR //Posizione Pinza - Metà ingombro - Offset sicurezza <= Ingombro colonna 
						(Mission^.YPick + IngombroOttimizzatoY_InTransito/2 + OffsetSicurezza_Y >= WorkFootprint^[6].Y) THEN //Posizione Pinza - Metà ingombro - Offset sicurezza <= Ingombro colonna 
							Pinza_InIngombroColonne_Transito := TRUE;
					ELSE
							Pinza_InIngombroColonne_Transito := FALSE;
					END_IF
			END_CASE		
			(* Se sono in ingombro nella posizione attuale o nella posizione di destinazione, devo andare fuori-ingombro con la Y *)
			IF (Pinza_InIngombroColonne_Attuale OR Pinza_InIngombroColonne_Destinazione OR Pinza_InIngombroColonne_Transito) AND AreaInLavoroPositivaNegativa THEN 
				IF (AsseXInFinestraDiRiposo AND AsseYInFinestraDiRiposo AND AsseJInFinestraDiRiposo) THEN //Se sono in finestra di riposo con tutti gli assi non devo andare fuori-ingombro con la Y
					FuoriIngombroYNecessarioTMP := FALSE;
				ELSE
					FuoriIngombroYNecessarioTMP := TRUE;
				END_IF
			ELSE
				FuoriIngombroYNecessarioTMP := FALSE;
			END_IF
		END_IF
		
	WAMANAGER_CICLO_DEPOSITO_PALL_END:
		CalcolaIngombro := TRUE;	
	
	WAMANAGER_CICLO_FALDA_VUOTI_INIT:
		CalcolaIngombro := TRUE;	
	
	WAMANAGER_CICLO_PRELIEVO_FALDA_VUOTI_RUN:
		IF CalcolaIngombro THEN
			CalcolaIngombro := FALSE;
			(* Definisco il tipo di area in cui si trova a lavorare il pallettizzatore *)
			AreaInLavoroPositiva := FALSE;
			AreaInLavoroNegativa := FALSE;
			AreaInLavoroPositivaNegativa := FALSE; 
			IF WorkArea^[Mission^.PPick].X >= (WorkFootprint^[5].X + WorkFootprint^[5].XDim) AND 	//se la piazzola di prelievo ha quota maggiore rispetto le colonne centrali
				ModuleAx_X^.Ax^.AxRef^.NcToPlc.ActPos >= (WorkFootprint^[5].X + WorkFootprint^[5].XDim)  THEN //Sono già nella campata positiva
					AreaInLavoroPositiva := TRUE;
			ELSIF WorkArea^[Mission^.PPick].X <= WorkFootprint^[5].X AND 	//se la piazzola di prelievo ha quota maggiore della piazzola di deposito e
				ModuleAx_X^.Ax^.AxRef^.NcToPlc.ActPos <= WorkFootprint^[5].X  THEN //Sono già nella campata negativa
					AreaInLavoroNegativa := TRUE;
			ELSE
				AreaInLavoroPositiva := FALSE;
				AreaInLavoroNegativa := FALSE;
				AreaInLavoroPositivaNegativa := TRUE;
			END_IF
			
			(**************************************************************************************************************************************************)
			(* Ingombro ottimizzato della pinza sul punto di prelievo *)
			(**************************************************************************************************************************************************)
			IngombroOttimizzatoX_InPuntoDiPrelievo := ABS(IngombroSuperficialePinzaMAX * SIN(deg_to_rad((ATAN(Larghezza/Lunghezza)*1/0.017+ Mission^.JPick))));
			IngombroOttimizzatoY_InPuntoDiPrelievo := ABS(IngombroSuperficialePinzaMAX * COS(deg_to_rad((ATAN(Larghezza/Lunghezza)*1/0.017+ Mission^.JPick))));
			(**************************************************************************************************************************************************)
			(* Ingombro ottimizzato della pinza sul punto di deposito *)
			(**************************************************************************************************************************************************)
			IngombroOttimizzatoX_InPuntoDiDeposito := ABS(IngombroSuperficialePinzaMAX * SIN(deg_to_rad((ATAN(Larghezza/Lunghezza)*1/0.017+ Mission^.JPlace))));
			IngombroOttimizzatoY_InPuntoDiDeposito := ABS(IngombroSuperficialePinzaMAX * COS(deg_to_rad((ATAN(Larghezza/Lunghezza)*1/0.017+ Mission^.JPlace))));
						
			(**************************************************************************************************************************************************)
			(**************************************************************************************************************************************************)
						
			(* Valuto la direzione della X *)
			DirezioneXPositiva := TFDirezioneAssePositiva(Posizione_Attuale:=ModuleAX_X^.Ax^.Status.ActPosition,Posizione_Finale:=Mission^.XPick);
			DirezioneXNegativa := NOT DirezioneXPositiva;
				
			(* Valuto se gli assi sono in finestra di prelievo *)
			AsseXInFinestraDiRiposo := TFAsseInFinestra(Posizione_Attuale:=ModuleAx_X^.Ax^.AxRef^.NcToPlc.ActPos,Posizione_Finale:=Mission^.XPick,FinestraDiControllo:=10);
			AsseYInFinestraDiRiposo := TFAsseInFinestra(Posizione_Attuale:=ModuleAx_Y^.Ax^.AxRef^.NcToPlc.ActPos,Posizione_Finale:=Mission^.YPick,FinestraDiControllo:=10);
			AsseJInFinestraDiRiposo := TFAsseInFinestra(Posizione_Attuale:=ModuleAx_J^.Ax^.AxRef^.NcToPlc.ActPos,Posizione_Finale:=Mission^.JPick,FinestraDiControllo:=5);
			(* Valuto se gli assi sono in finestra di destinazione *)
			AsseXInFinestraDiDestinazione := TFAsseInFinestra(Posizione_Attuale:=ModuleAx_X^.Ax^.AxRef^.NcToPlc.ActPos,Posizione_Finale:=Mission^.XPick,FinestraDiControllo:=10);
			AsseYInFinestraDiDestinazione := TFAsseInFinestra(Posizione_Attuale:=ModuleAx_Y^.Ax^.AxRef^.NcToPlc.ActPos,Posizione_Finale:=Mission^.YPick,FinestraDiControllo:=10);
			AsseJInFinestraDiDestinazione := TFAsseInFinestra(Posizione_Attuale:=ModuleAx_J^.Ax^.AxRef^.NcToPlc.ActPos,Posizione_Finale:=Mission^.JPick,FinestraDiControllo:=5);
			
			(**************************************************************************************************************************************************)
			(* Ingombro MASSIMO della pinza durante il transito *)
			(**************************************************************************************************************************************************)
			//Calcolo ingombro attuale
			IngombroOttimizzatoX_InTransito := ABS(IngombroSuperficialePinzaMAX * SIN(deg_to_rad((ATAN(Larghezza/Lunghezza)*1/0.017+ ModuleAx_J^.Ax^.AxRef^.NcToPlc.ActPos)))); //Ingombro Attuale direzione X
			IngombroOttimizzatoY_InTransito := ABS(IngombroSuperficialePinzaMAX * COS(deg_to_rad((ATAN(Larghezza/Lunghezza)*1/0.017+ ModuleAx_J^.Ax^.AxRef^.NcToPlc.ActPos)))); //Ingombro Attuale direzione Y		
			IF NOT AsseJInFinestraDiDestinazione THEN
				IF REAL_TO_INT(ModuleAx_J^.Ax^.AxRef^.NcToPlc.ActPos) <= REAL_TO_INT(Mission^.JPick) THEN
					FOR Angolo := REAL_TO_INT(ModuleAx_J^.Ax^.AxRef^.NcToPlc.ActPos) TO REAL_TO_INT(Mission^.JPick)  DO
						IF IngombroOttimizzatoX_InTransito < ABS(IngombroSuperficialePinzaMAX * SIN(deg_to_rad((ATAN(Larghezza/Lunghezza)*1/0.017+ Angolo)))) THEN
							IngombroOttimizzatoX_InTransito := ABS(IngombroSuperficialePinzaMAX * SIN(deg_to_rad((ATAN(Larghezza/Lunghezza)*1/0.017+ Angolo)))) ;
						END_IF
						IF IngombroOttimizzatoY_InTransito < ABS(IngombroSuperficialePinzaMAX * COS(deg_to_rad((ATAN(Larghezza/Lunghezza)*1/0.017+ Angolo)))) THEN
							IngombroOttimizzatoY_InTransito := ABS(IngombroSuperficialePinzaMAX * COS(deg_to_rad((ATAN(Larghezza/Lunghezza)*1/0.017+ Angolo))));
						END_IF
					END_FOR
				END_IF
			END_IF
		
			(* Valutazione colonne in base al verso del pallettizzatore *)
			CASE VERSO_PALLETTIZZATORE OF
				PALLETTIZZATORE_DX:	// Colonna 6:DX, 5:SX
					(* Valuto la posizione attuale *)
					IF (ModuleAX_Y^.Ax^.Status.ActPosition - IngombroY/2 - OffsetSicurezza_Y <= WorkFootprint^[6].Y) OR //Posizione Pinza - Metà ingombro - Offset sicurezza <= Ingombro colonna 
						(ModuleAX_Y^.Ax^.Status.ActPosition + IngombroY/2 + OffsetSicurezza_Y >= WorkFootprint^[5].Y) THEN //Posizione Pinza - Metà ingombro - Offset sicurezza <= Ingombro colonna 
							Pinza_InIngombroColonne_Attuale := TRUE;
					ELSE
							Pinza_InIngombroColonne_Attuale := FALSE;
					END_IF
					(* Valuto la posizione futura - Missione di prelievo *)
					IF (Mission^.YPick - IngombroOttimizzatoX_InPuntoDiPrelievo/2 - OffsetSicurezza_Y <= WorkFootprint^[6].Y) OR //Posizione Pinza - Metà ingombro - Offset sicurezza <= Ingombro colonna 
						(Mission^.YPick + IngombroOttimizzatoX_InPuntoDiPrelievo/2 + OffsetSicurezza_Y >= WorkFootprint^[5].Y) THEN //Posizione Pinza - Metà ingombro - Offset sicurezza <= Ingombro colonna 
							Pinza_InIngombroColonne_Destinazione := TRUE;
					ELSE
							Pinza_InIngombroColonne_Destinazione := FALSE;
					END_IF
					
					(* Valuto la posizione futura - Missione di Deposito *)
					IF (Mission^.YPick - IngombroOttimizzatoX_InPuntoDiDeposito/2 - OffsetSicurezza_Y <= WorkFootprint^[6].Y) OR //Posizione Pinza - Metà ingombro - Offset sicurezza <= Ingombro colonna 
						(Mission^.YPick + IngombroOttimizzatoX_InPuntoDiDeposito/2 + OffsetSicurezza_Y >= WorkFootprint^[5].Y) THEN //Posizione Pinza - Metà ingombro - Offset sicurezza <= Ingombro colonna 
							Pinza_InIngombroColonne_Destinazione := TRUE;
					ELSE
							Pinza_InIngombroColonne_Destinazione := FALSE;
					END_IF
					
					(* Valuto la posizione attuale Y e la posizione di destinazione Y e l'ingombro massimo che posso avere durante il transito *)
					IF (Mission^.YPick - IngombroOttimizzatoY_InTransito/2 - OffsetSicurezza_Y <= WorkFootprint^[6].Y) OR //Posizione Pinza - Metà ingombro - Offset sicurezza <= Ingombro colonna 
						(Mission^.YPick + IngombroOttimizzatoY_InTransito/2 + OffsetSicurezza_Y >= WorkFootprint^[5].Y) THEN //Posizione Pinza - Metà ingombro - Offset sicurezza <= Ingombro colonna 
							Pinza_InIngombroColonne_Transito := TRUE;
					ELSE
							Pinza_InIngombroColonne_Transito := FALSE;
					END_IF
						
				PALLETTIZZATORE_SX: // Colonna 6:SX, 5:DX
					(* Valuto la posizione attuale *)
					IF (ModuleAX_Y^.Ax^.Status.ActPosition - IngombroY/2 - OffsetSicurezza_Y <= WorkFootprint^[5].Y) OR //Posizione Pinza - Metà ingombro - Offset sicurezza <= Ingombro colonna 
						(ModuleAX_Y^.Ax^.Status.ActPosition + IngombroY/2 + OffsetSicurezza_Y >= WorkFootprint^[6].Y) THEN //Posizione Pinza - Metà ingombro - Offset sicurezza <= Ingombro colonna 
							Pinza_InIngombroColonne_Attuale := TRUE;
					ELSE
							Pinza_InIngombroColonne_Attuale := FALSE;
					END_IF
					(* Valuto la posizione futura - Missione di prelievo *)
					IF (Mission^.YPick - IngombroOttimizzatoX_InPuntoDiPrelievo/2 - OffsetSicurezza_Y <= WorkFootprint^[5].Y) OR //Posizione Pinza - Metà ingombro - Offset sicurezza <= Ingombro colonna 
						(Mission^.YPick + IngombroOttimizzatoX_InPuntoDiPrelievo/2 + OffsetSicurezza_Y >= WorkFootprint^[6].Y) THEN //Posizione Pinza - Metà ingombro - Offset sicurezza <= Ingombro colonna 
							Pinza_InIngombroColonne_Destinazione := TRUE;
					ELSE
							Pinza_InIngombroColonne_Destinazione := FALSE;
					END_IF
					
					(* Valuto la posizione futura - Missione di Deposito *)
					IF (Mission^.YPick - IngombroOttimizzatoX_InPuntoDiDeposito/2 - OffsetSicurezza_Y <= WorkFootprint^[5].Y) OR //Posizione Pinza - Metà ingombro - Offset sicurezza <= Ingombro colonna 
						(Mission^.YPick + IngombroOttimizzatoX_InPuntoDiDeposito/2 + OffsetSicurezza_Y >= WorkFootprint^[6].Y) THEN //Posizione Pinza - Metà ingombro - Offset sicurezza <= Ingombro colonna 
							Pinza_InIngombroColonne_Destinazione := TRUE;
					ELSE
							Pinza_InIngombroColonne_Destinazione := FALSE;
					END_IF
					
